// TwinCAT 3 PLC project CamerasTCP_Drivers
// ProgramVersion: 3.1.4026.19
// libraries:
//   Tc2_SerialCom, * (Beckhoff Automation GmbH)
//   Tc2_Standard, * (Beckhoff Automation GmbH)
//   Tc2_System, * (Beckhoff Automation GmbH)
//   Tc2_TcpIp, * (Beckhoff Automation GmbH)
//   Tc2_Utilities, * (Beckhoff Automation GmbH)
// project tree:
//   DUTs/ E_STRING_ExtrMode.TcDUT (not stored), E_TCPIP_RequescCommand.TcDUT, E_TCPIP_SEND_STATE.TcDUT, E_TCPIP_State.TcDUT, T_LongSTRING.TcDUT (not stored)
//   DUTs/NewModel/CameraImage/ E_CAMERA_State.TcDUT, ST_CAMERA_CodeData.TcDUT, ST_CAMERA_ImageData.TcDUT, ST_CAMERA_TriggerID.TcDUT, ST_GS1_AI.TcDUT
//   DUTs/NewModel/ E_CAMERA_Name.TcDUT, ST_CAMERA_Evaluation.TcDUT
//   DUTs/NewModel/Main Struct/Config/ E_CAMERA_CodeType.TcDUT, E_CAMERA_DeviceType.TcDUT, E_CAMERA_Vendor.TcDUT, ST_CAMERA_Options.TcDUT
//   DUTs/NewModel/Main Struct/Control/ ST_CAMERA_BrowseCtrl.TcDUT, ST_CAMERA_Mapping.TcDUT
//   DUTs/NewModel/Main Struct/Status/ E_CAMERA_Status.TcDUT, ST_CAMERA_BrowserStatus.TcDUT, ST_CAMERA_IN.TcDUT, ST_CAMERA_OpState.TcDUT, ST_CAMERA_OUT.TcDUT, ST_CAMERA_Performance.TcDUT
//   DUTs/NewModel/Main Struct/ ST_CAMERA_Config.TcDUT, ST_CAMERA_Ctrl.TcDUT, ST_CAMERA_Status.TcDUT
//   DUTs/Test_DUTs/ ST_DuplicateInfo.TcDUT (not stored), ST_LAB_CaseData.TcDUT, ST_LAB_OuterData.TcDUT, ST_LAB_PackData.TcDUT (not stored)
//   DUTs/USED/ E_SCANNER_CodeType.TcDUT (not stored), E_SCANNER_DeviceType.TcDUT (not stored), E_SCANNER_State.TcDUT (not stored), E_SCANNER_Vendor.TcDUT (not stored), ST_SCANNER.TcDUT, ST_SCANNER_ApplicationIdentifier.TcDUT (not stored), ST_SCANNER_CameraMap.TcDUT (not stored), ST_SCANNER_CodeData.TcDUT (not stored), ST_SCANNER_Config.TcDUT (not stored), ST_SCANNER_Evaluation.TcDUT (not stored), ST_SCANNER_ImageData.TcDUT (not stored), ST_SCANNER_ManualCtrl.TcDUT (not stored), ST_SCANNER_OpState.TcDUT (not stored), ST_SCANNER_Options.TcDUT (not stored), ST_SCANNER_Performance.TcDUT (not stored), ST_SCANNER_TriggerID.TcDUT (not stored)
//   GVLs/ gConstants.TcGVL (not stored), GVL.TcGVL, GVL_HIKROBOT_COMMANDS.TcGVL (not stored), GVL_test.TcGVL
//   / PlcTask.TcTTO
//   POUs/Addtionals/ FB_PulseGenerator_Sync.TcPOU (not stored), PRG_ButtonsHandler.TcPOU
//   POUs/CAMERAS/ FB_SCANNER_HikrobotEXT.TcPOU, F_CREATE_MESSAGE.TcPOU (not stored)
//   POUs/ MAIN.TcPOU, PRG_HikrobotHandler.TcPOU
//   POUs/NewModel/ FB_CAMERA_Omron.TcPOU, FB_CAMERA_HIKROBOT.TcPOU
//   POUs/SOFTWARE_lib/TCP FBs/ FB_TCP_ClientPortCtrl.TcPOU, FB_TCP_ClientPortCtrl_V2.TcPOU, FB_TCP_CloseAllPorts.TcPOU, FB_TCP_ReceiveData_V2.TcPOU, FB_TCP_ReceiveLongString.TcPOU (not stored), FB_TCP_ReceiveString.TcPOU (not stored), FB_TCP_SendData.TcPOU, FB_TCP_ServerPortCtrl.TcPOU
//   POUs/StringFBs/ FB_ExtractAnyString.TcPOU
//   POUs/Tests/ FB_FIND_OuterDuplicates.TcPOU, IO_logic.TcPOU (not stored), Outer_IN_Case_Duplicat.TcPOU, PRG_Test.TcPOU
// real-time tasks:
//   TASK PlcTask: cycle T#10ms, priority 20, ADS port 350
// motion (NC):
//   TASK NC-Task 1 SAF: cycle T#2ms, priority 4, ADS port 501
//   TASK NC-Task 1 SVB: cycle T#10ms, priority 8, ADS port 511
//   AXIS Axis 1 (id 1)
//     OtherSettings: AllowMotionCmdToSlave=true
//     encoder EncType=4
//       EncPara: MaxCount=#x0000ffff
//         Inc: RefSoftSyncMask=#x0000ffff
//     drive DrvType=24
//       Analog: TorqueSetpointScale=10, ScaleFactorActTorque=0.1
//       TimeComp: TaskDelayCycles=1
//     controller CtrType=1
//       CtrPara: PriorControlFactor=1
//         Observer: BandWidth=20
//   AXIS Axis 2 (id 2)
//     OtherSettings: AllowMotionCmdToSlave=true
//     encoder EncType=4
//       EncPara: MaxCount=#x0000ffff
//         Inc: RefSoftSyncMask=#x0000ffff
//     drive DrvType=24
//       Analog: TorqueSetpointScale=10, ScaleFactorActTorque=0.1
//       TimeComp: TaskDelayCycles=1
//     controller CtrType=1
//       CtrPara: PriorControlFactor=1
//         Observer: BandWidth=20
//   AXIS Axis 3 (id 3)
//     OtherSettings: AllowMotionCmdToSlave=true
//     encoder EncType=19
//       EncPara: MaxCount=#xffffffff
//     drive DrvType=16
//       DrvPara: MaxCount=#xffffffff
//         Analog: TorqueSetpointScale=10, ScaleFactorActTorque=0.1
//         TimeComp: TaskDelayCycles=1
//     controller CtrType=1
//       CtrPara: PriorControlFactor=1
//         Observer: BandWidth=20
//   AXIS Axis 4 (id 4)
//     OtherSettings: AllowMotionCmdToSlave=true
//     encoder EncType=4
//       EncPara: MaxCount=#x0000ffff
//         Inc: RefSoftSyncMask=#x0000ffff
//     drive DrvType=24
//       Analog: TorqueSetpointScale=10, ScaleFactorActTorque=0.1
//       TimeComp: TaskDelayCycles=1
//     controller CtrType=1
//       CtrPara: PriorControlFactor=1
//         Observer: BandWidth=20
//   AXIS Axis 5 (id 5)
//     OtherSettings: AllowMotionCmdToSlave=true
//     encoder EncType=4
//       EncPara: MaxCount=#x0000ffff
//         Inc: RefSoftSyncMask=#x0000ffff
//     drive DrvType=24
//       Analog: TorqueSetpointScale=10, ScaleFactorActTorque=0.1
//       TimeComp: TaskDelayCycles=1
//     controller CtrType=1
//       CtrPara: PriorControlFactor=1
//         Observer: BandWidth=20
//   AXIS Axis 6 (id 6)
//     OtherSettings: AllowMotionCmdToSlave=true
//     encoder EncType=19
//       EncPara: MaxCount=#xffffffff
//     drive DrvType=16
//       DrvPara: MaxCount=#xffffffff
//         Analog: TorqueSetpointScale=10, ScaleFactorActTorque=0.1
//         TimeComp: TaskDelayCycles=1
//     controller CtrType=1
//       CtrPara: PriorControlFactor=1
//         Observer: BandWidth=20
//   AXIS Axis 7 (id 7)
//     OtherSettings: AllowMotionCmdToSlave=true
//     encoder EncType=4
//       EncPara: MaxCount=#x0000ffff
//         Inc: RefSoftSyncMask=#x0000ffff
//     drive DrvType=24
//       Analog: TorqueSetpointScale=10, ScaleFactorActTorque=0.1
//       TimeComp: TaskDelayCycles=1
//     controller CtrType=1
//       CtrPara: PriorControlFactor=1
//         Observer: BandWidth=20
//   AXIS Axis 8 (id 8)
//     OtherSettings: AllowMotionCmdToSlave=true
//     encoder EncType=4
//       EncPara: MaxCount=#x0000ffff
//         Inc: RefSoftSyncMask=#x0000ffff
//     drive DrvType=24
//       Analog: TorqueSetpointScale=10, ScaleFactorActTorque=0.1
//       TimeComp: TaskDelayCycles=1
//     controller CtrType=1
//       CtrPara: PriorControlFactor=1
//         Observer: BandWidth=20
//   AXIS Axis 9 (id 9)
//     OtherSettings: AllowMotionCmdToSlave=true
//     encoder EncType=19
//       EncPara: MaxCount=#xffffffff
//     drive DrvType=16
//       DrvPara: MaxCount=#xffffffff, DriveControlDWord=#x00020000
//         Analog: TorqueSetpointScale=10, ScaleFactorActTorque=0.1
//         TimeComp: TaskDelayCycles=1
//     controller CtrType=1
//       CtrPara: PriorControlFactor=1
//         Observer: BandWidth=20
//   AXIS Axis 10 (id 10)
//     OtherSettings: AllowMotionCmdToSlave=true
//     encoder EncType=4
//       EncPara: MaxCount=#x0000ffff
//         Inc: RefSoftSyncMask=#x0000ffff
//     drive DrvType=24
//       Analog: TorqueSetpointScale=10, ScaleFactorActTorque=0.1
//       TimeComp: TaskDelayCycles=1
//     controller CtrType=1
//       CtrPara: PriorControlFactor=1
//         Observer: BandWidth=20
//   AXIS Axis 11 (id 11)
//     OtherSettings: AllowMotionCmdToSlave=true
//     encoder EncType=4
//       EncPara: MaxCount=#x0000ffff
//         Inc: RefSoftSyncMask=#x0000ffff
//     drive DrvType=24
//       Analog: TorqueSetpointScale=10, ScaleFactorActTorque=0.1
//       TimeComp: TaskDelayCycles=1
//     controller CtrType=1
//       CtrPara: PriorControlFactor=1
//         Observer: BandWidth=20
//   AXIS Axis 12 (id 12)
//     OtherSettings: AllowMotionCmdToSlave=true
//     encoder EncType=19
//       EncPara: MaxCount=#xffffffff
//     drive DrvType=16
//       DrvPara: MaxCount=#xffffffff
//         Analog: TorqueSetpointScale=10, ScaleFactorActTorque=0.1
//         TimeComp: TaskDelayCycles=1
//     controller CtrType=1
//       CtrPara: PriorControlFactor=1
//         Observer: BandWidth=20
// I/O:
//   DEVICE Device 1 (EtherCAT) (disabled), AmsNetId 192.168.1.11.2.1
//     Term 1 (EK1100)
//     Term 9 (EK1100) [EK1100 EtherCAT Coupler (2A E-Bus)]
//       Term 10 (EL7031-0030)
//       Term 11 (EL6070-0033)
//       Term 12 (EL7031-0030)
//       Term 17 (EL9011)
//     Term 13 (EK1818)
// variable links:
//   (this object) <-> Device 1 (EtherCAT)/Term 9 (EK1100)/Term 10 (EL7031-0030)
//     Drive/Inputs/In/nState1 @bit 3 <-> STM Status/Status/Error
//     Drive/Inputs/In/nState1 @bit 5 <-> STM Status/Status/Moving negative
//     Drive/Inputs/In/nState1 @bit 4 <-> STM Status/Status/Moving positive
//     Drive/Inputs/In/nState1 @bit 1 <-> STM Status/Status/Ready
//     Drive/Inputs/In/nState1 <-> STM Status/Status/Ready to enable
//     Drive/Inputs/In/nState1 @bit 6 <-> STM Status/Status/Torque reduced
//     Drive/Inputs/In/nState1 @bit 2 <-> STM Status/Status/Warning
//     Drive/Inputs/In/nState2 @bit 3 <-> STM Status/Status/Digital input 1
//     Drive/Inputs/In/nState2 @bit 4 <-> STM Status/Status/Digital input 2
//     Drive/Inputs/In/nState2 @bit 5 <-> STM Status/Status/Sync error
//     Drive/Inputs/In/nState2 @bit 7 <-> STM Status/Status/TxPDO Toggle
//     Drive/Inputs/In/nState4 @bit 1 <-> WcState/InputToggle
//     Drive/Inputs/In/nState4 <-> WcState/WcState
//     Drive/Outputs/Out/nCtrl1 <-> STM Control/Control/Enable
//     Drive/Outputs/Out/nCtrl1 @bit 2 <-> STM Control/Control/Reduce torque
//     Drive/Outputs/Out/nCtrl1 @bit 1 <-> STM Control/Control/Reset
//     Drive/Outputs/Out/nDataOut2[0] <-> STM Velocity/Velocity
//     Enc/Inputs/In/nDataIn1[0] <-> ENC Status compact/Counter value
//     Enc/Inputs/In/nDataIn2[0] <-> ENC Status compact/Latch value
//     Enc/Inputs/In/nState1 @bit 4 <-> ENC Status compact/Status/Counter overflow
//     Enc/Inputs/In/nState1 @bit 3 <-> ENC Status compact/Status/Counter underflow
//     Enc/Inputs/In/nState1 @bit 1 <-> ENC Status compact/Status/Latch extern valid
//     Enc/Inputs/In/nState1 @bit 2 <-> ENC Status compact/Status/Set counter done
//     Enc/Inputs/In/nState2 @bit 4 <-> ENC Status compact/Status/Status of extern latch
//     Enc/Inputs/In/nState2 @bit 5 <-> ENC Status compact/Status/Sync error
//     Enc/Inputs/In/nState2 @bit 7 <-> ENC Status compact/Status/TxPDO Toggle
//     Enc/Inputs/In/nState4 @bit 1 <-> WcState/InputToggle
//     Enc/Inputs/In/nState4 <-> WcState/WcState
//     Enc/Outputs/Out/nCtrl1 @bit 3 <-> ENC Control compact/Control/Enable latch extern on negative edge
//     Enc/Outputs/Out/nCtrl1 @bit 1 <-> ENC Control compact/Control/Enable latch extern on positive edge
//     Enc/Outputs/Out/nCtrl1 @bit 2 <-> ENC Control compact/Control/Set counter
//     Enc/Outputs/Out/nDataOut1[0] <-> ENC Control compact/Set counter value
//   (this object) <-> Device 1 (EtherCAT)/Term 9 (EK1100)/Term 12 (EL7031-0030)
//     Drive/Inputs/In/nState1 @bit 3 <-> STM Status/Status/Error
//     Drive/Inputs/In/nState1 @bit 5 <-> STM Status/Status/Moving negative
//     Drive/Inputs/In/nState1 @bit 4 <-> STM Status/Status/Moving positive
//     Drive/Inputs/In/nState1 @bit 1 <-> STM Status/Status/Ready
//     Drive/Inputs/In/nState1 <-> STM Status/Status/Ready to enable
//     Drive/Inputs/In/nState1 @bit 6 <-> STM Status/Status/Torque reduced
//     Drive/Inputs/In/nState1 @bit 2 <-> STM Status/Status/Warning
//     Drive/Inputs/In/nState2 @bit 3 <-> STM Status/Status/Digital input 1
//     Drive/Inputs/In/nState2 @bit 4 <-> STM Status/Status/Digital input 2
//     Drive/Inputs/In/nState2 @bit 5 <-> STM Status/Status/Sync error
//     Drive/Inputs/In/nState2 @bit 7 <-> STM Status/Status/TxPDO Toggle
//     Drive/Inputs/In/nState4 @bit 1 <-> WcState/InputToggle
//     Drive/Inputs/In/nState4 <-> WcState/WcState
//     Drive/Outputs/Out/nCtrl1 <-> STM Control/Control/Enable
//     Drive/Outputs/Out/nCtrl1 @bit 2 <-> STM Control/Control/Reduce torque
//     Drive/Outputs/Out/nCtrl1 @bit 1 <-> STM Control/Control/Reset
//     Drive/Outputs/Out/nDataOut2[0] <-> STM Velocity/Velocity
//     Enc/Inputs/In/nDataIn1[0] <-> ENC Status compact/Counter value
//     Enc/Inputs/In/nDataIn2[0] <-> ENC Status compact/Latch value
//     Enc/Inputs/In/nState1 @bit 4 <-> ENC Status compact/Status/Counter overflow
//     Enc/Inputs/In/nState1 @bit 3 <-> ENC Status compact/Status/Counter underflow
//     Enc/Inputs/In/nState1 @bit 1 <-> ENC Status compact/Status/Latch extern valid
//     Enc/Inputs/In/nState1 @bit 2 <-> ENC Status compact/Status/Set counter done
//     Enc/Inputs/In/nState2 @bit 4 <-> ENC Status compact/Status/Status of extern latch
//     Enc/Inputs/In/nState2 @bit 5 <-> ENC Status compact/Status/Sync error
//     Enc/Inputs/In/nState2 @bit 7 <-> ENC Status compact/Status/TxPDO Toggle
//     Enc/Inputs/In/nState4 @bit 1 <-> WcState/InputToggle
//     Enc/Inputs/In/nState4 <-> WcState/WcState
//     Enc/Outputs/Out/nCtrl1 @bit 3 <-> ENC Control compact/Control/Enable latch extern on negative edge
//     Enc/Outputs/Out/nCtrl1 @bit 1 <-> ENC Control compact/Control/Enable latch extern on positive edge
//     Enc/Outputs/Out/nCtrl1 @bit 2 <-> ENC Control compact/Control/Set counter
//     Enc/Outputs/Out/nDataOut1[0] <-> ENC Control compact/Set counter value
//   (this object) <-> Device 1 (EtherCAT)/Term 13 (EK1818)/Term 14 (EL7211-9014)
//     Drive/Inputs/In/nDcOutputTime <-> InfoData/DcOutputShift
//     Drive/Inputs/In/nState1 <-> DRV Statusword/Statusword
//     Drive/Inputs/In/nState2 <-> DRV Statusword/Statusword @bit 8
//     Drive/Inputs/In/nState4 @bit 1 <-> WcState/InputToggle
//     Drive/Inputs/In/nState4 <-> WcState/WcState
//     Drive/Outputs/Out/nCtrl1 <-> DRV Controlword/Controlword
//     Drive/Outputs/Out/nCtrl2 <-> DRV Controlword/Controlword @bit 8
//     Drive/Outputs/Out/nDataOut2 <-> DRV Target velocity/Target velocity
//     Enc/Inputs/In/nDataIn1 <-> FB Position/Position
//     Enc/Inputs/In/nDcInputTime <-> InfoData/DcInputShift
//     Enc/Inputs/In/nState4 @bit 1 <-> WcState/InputToggle
//     Enc/Inputs/In/nState4 <-> WcState/WcState

CONFIGURATION CamerasTCP_Drivers
    RESOURCE PLC ON TwinCAT3
        TASK PlcTask(INTERVAL := T#10ms, PRIORITY := 20);
        PROGRAM MAIN WITH PlcTask : MAIN;
    END_RESOURCE
END_CONFIGURATION

// ---- DUTs/E_TCPIP_RequescCommand.TcDUT
{attribute 'qualified_only'}
{attribute 'strict'}
{attribute 'to_string'}
TYPE E_TCPIP_RequescCommand :
(
	NONE,					(* No request to send *)
	SetRunMode,				(* Set run mode, 0 - Normal, 1 - Raw, 2 - Test *)
	SetAcq,					(* Set acquisition mode, 0 - Stop acq, 1 - Start acq *)
	GetUserCur,
	HeartbeatCheck			
);
END_TYPE

// ---- DUTs/E_TCPIP_SEND_STATE.TcDUT
{attribute 'qualified_only'}
{attribute 'strict'}
{attribute 'to_string'}
TYPE E_TCPIP_SEND_STATE :
(
	IDLE,
	CONNECT,
	SEND,
	RECEIVE,
	DISCONNECT,
	DONE,
	CONN_RESET,
	HEARTBEAT_CHECK,
	ERROR
);
END_TYPE

// ---- DUTs/E_TCPIP_State.TcDUT
{attribute 'qualified_only'}
{attribute 'strict'}
{attribute 'to_string'}
TYPE E_TCPIP_State :
(
	E_TCPIP_IDLE,
	E_TCPIP_CONNECT,
	E_TCPIP_SEND,
	E_TCPIP_RECEIVE,
	E_TCPIP_DISCONNECT,
	E_TCPIP_CLOSEALL,
	E_TCPIP_DONE
);
END_TYPE

// ---- DUTs/NewModel/CameraImage/E_CAMERA_State.TcDUT
{attribute 'qualified_only'}
{attribute 'strict'}
TYPE E_CAMERA_State :
(
	IDLE,
	CONNECT,
	SEND,
	RECEIVE,
	DISCONNECT,
	//CHECKOS,
	BROWSEDIAG,
	BROWSELIVE,
	IMAGE,
	DECODE,
	HEARTBEAT,
	DONE
);
END_TYPE

// ---- DUTs/NewModel/CameraImage/ST_CAMERA_CodeData.TcDUT
TYPE ST_CAMERA_CodeData :
STRUCT
	nScannerIndex		: INT;			(* scanner index when an array of scanners is used *)
	sDataString			: T_MaxString;	(* data string read from code *)
	eCodeType			: E_CAMERA_CodeType;	(* code type *)
	fOverallGrade		: LREAL;		(* overall grade of code *)
	fXPos				: LREAL;		(* X position of centre of code *)
	fYPos				: LREAL;		(* Y position of centre of code *)
	fAngle				: LREAL;		(* angle of code *)
	fCellSize			: LREAL;		(* cell size *)
	fSymbolContrast		: LREAL;		(* symbol contrast *)
	nEvaluation			: INT;			(* general code quality evaluatio*)
	fUnusedErrCorr		: LREAL;		(* unused error correction *)
	nProgramNo			: BYTE;			(* program number *)
END_STRUCT
END_TYPE

// ---- DUTs/NewModel/CameraImage/ST_CAMERA_ImageData.TcDUT
TYPE ST_CAMERA_ImageData :
STRUCT
	nCodesRead		: INT;
	tScanTime		: TIME;		(* image cycle time (including image acquisition time and decode time) *)
	sDecodeStatus	: T_MaxString;
	stTriggerID		: ST_CAMERA_TriggerID;
	aCodeData		: ARRAY[1..cMAX_CAMERA_PROG_NUMBER] OF ST_CAMERA_CodeData;
END_STRUCT
END_TYPE

// ---- DUTs/NewModel/CameraImage/ST_CAMERA_TriggerID.TcDUT
TYPE ST_CAMERA_TriggerID :
STRUCT
	nTriggerID			: UDINT;
	nScanNo				: INT := 1;
	nScannerIndex		: INT := 1;
END_STRUCT
END_TYPE

// ---- DUTs/NewModel/CameraImage/ST_GS1_AI.TcDUT
TYPE ST_GS1_AI :
STRUCT
	sAI			: STRING(4);
	bFixed		: BOOL;
	nLength		: UINT;
END_STRUCT
END_TYPE

// ---- DUTs/NewModel/E_CAMERA_Name.TcDUT
{attribute 'qualified_only'}
//{attribute 'strict'}
TYPE E_CAMERA_Name :
(
	CAM01		:= 1,
	CAM02		:= 2,
	CAM03		:= 3,
	CAM04		:= 4,
	CAM05		:= 5,
	CAM06		:= 6,
	CAM07		:= 7,
	CAM08		:= 8,
	CAM09		:= 9,
	CAM10		:= 10,
	CAM11		:= 11,
	CAM12		:= 12
);
END_TYPE

// ---- DUTs/NewModel/Main Struct/Config/E_CAMERA_CodeType.TcDUT
{attribute 'qualified_only'}
//{attribute 'strict'}
TYPE E_CAMERA_CodeType :
(
	NONE 		:= 0,
	OCR			:= 7,
	DATAMARTIX	:= 10,
	QR			:= 11,
	DOTCODE		:= 14,
	CODE128		:= 20,
	ITF14		:= 24,
	EAN13		:= 27,
	EAN8		:= 28,
	UNKNOWN		:= 99
);
END_TYPE

// ---- DUTs/NewModel/Main Struct/Config/E_CAMERA_DeviceType.TcDUT
{attribute 'qualified_only'}
//{attribute 'strict'}
TYPE E_CAMERA_DeviceType :    (*tAcquisitionTime - to be secured*)
(
	NONE,
	MV420_F,			//F -> Full resolution
	MV420_H,			//H -> Half resolution
	MV440SR_F,
	MV440SR_H,
	MV440HR_F,
	MV440HR_H,
	MV440UR_F,
	MV440UR_H,
	MV540S_F,
	MV540S_H,
	MV540H_F,
	MV540H_H,
	MV560U_F,
	MV560U_H,
	V430F	(*Omron*)

);
END_TYPE

// ---- DUTs/NewModel/Main Struct/Config/E_CAMERA_Vendor.TcDUT
{attribute 'qualified_only'}
{attribute 'strict'}
TYPE E_CAMERA_Vendor :
(
	SIEMENS		:= 1,
	OMRON 		:= 2,
	KEYENCE		:= 3,
	COGNEX		:= 4,
	HIKROBOT	:= 5
);
END_TYPE

// ---- DUTs/NewModel/Main Struct/Config/ST_CAMERA_Options.TcDUT
TYPE ST_CAMERA_Options :
STRUCT
	eScannerType			: E_CAMERA_DeviceType;
	eExpectedType			: E_CAMERA_CodeType;
	bUseExternalLight		: BOOL;
	nLightingIntensity		: INT;
	nDisplayDelayConfig		: BOOL;

	nImageBuffer			: INT := 1;
	nExpectedResp			: INT := 1;
	
	aCameraWarningLevel		: INT := 90;
	sFC1ReplacmentChar		: T_Char;
END_STRUCT
END_TYPE

// ---- DUTs/NewModel/Main Struct/Control/ST_CAMERA_BrowseCtrl.TcDUT
TYPE ST_CAMERA_BrowseCtrl :
STRUCT
	bBrowseLive			: BOOL;	
	bBrowseDiag			: BOOL;
END_STRUCT
END_TYPE

// ---- DUTs/NewModel/Main Struct/Control/ST_CAMERA_Mapping.TcDUT
TYPE ST_CAMERA_Mapping :
STRUCT
	nIndex				: INT;
	nReqProgram			: BYTE;
	aPackPos			: ARRAY[1..5, 1..cMAX_CAMERA_PROG_NUMBER] OF BYTE;
	aTargetBuffer		: ARRAY[1..5] OF BYTE;

END_STRUCT
END_TYPE

// ---- DUTs/NewModel/Main Struct/Status/E_CAMERA_Status.TcDUT
{attribute 'qualified_only'}
{attribute 'strict'}

TYPE E_CAMERA_Status :
(
			
	DIABLED 		:= 0,		//0 = Grey, disabled OR offline
	CONFIG			:= 1,		//1 = Blue, configuration mode active
	ALARM			:= 2,		//2 = Red, alarm active or comms loss
	EXTERNALOFF		:= 3,		//3 = Orange, external condition off
	WARNING			:= 4,		//4 = Yellow, warning active
	OERATIONAL		:= 5		//5 = Green, operational	
);
END_TYPE

// ---- DUTs/NewModel/Main Struct/Status/ST_CAMERA_BrowserStatus.TcDUT
TYPE ST_CAMERA_BrowserStatus :
STRUCT
	bBrowseLiveActive			: BOOL;	
	bBrowseDiagActive			: BOOL;
END_STRUCT
END_TYPE

// ---- DUTs/NewModel/Main Struct/Status/ST_CAMERA_IN.TcDUT
TYPE ST_CAMERA_IN :
STRUCT
	stTriggerID			: ST_CAMERA_TriggerID;	
	stBrowserStatus		: ST_CAMERA_BrowserStatus;
	
END_STRUCT
END_TYPE

// ---- DUTs/NewModel/Main Struct/Status/ST_CAMERA_OpState.TcDUT
TYPE ST_CAMERA_OpState :
STRUCT
	nStatusByte			: BYTE;
	nErrorCode			: UDINT;
	nWarningCode		: UDINT;

	bAcceptTrigger		: BOOL;
	bCodeChangeActive	: BOOL;
	nActiveTriggers		: INT;

	bTCPComsLockedUp	: BOOL;

END_STRUCT
END_TYPE

// ---- DUTs/NewModel/Main Struct/Status/ST_CAMERA_OUT.TcDUT
TYPE ST_CAMERA_OUT :
STRUCT
	bDone								: BOOL;			(* TRUE = code scan complete *)
	bBusy								: BOOL;			(* TRUE = code scan in progress *)
	bError								: BOOL;			(* TRUE = code scan error *)

	bReady								: BOOL;			(* TRUE = scanner port connected *)
	bEnableActive						: BOOL;
	nTriggerCounter						: UDINT;

	nActiveProgram						: BYTE;			(* active program *)
	stOpState							: ST_CAMERA_OpState;	(* operating state values *)
	
	sCodeStatus							: T_MaxString;				(* image status string *)
	sCurrentCodeRead					: T_MaxString;
	aLast10CodesRead					: ARRAY[1..10]  OF T_MaxString;
	stImageData							: ST_CAMERA_ImageData;		(* image data structure *)
	stReadPerformance					: ST_CAMERA_Performance;
	
	eSocketState						: E_SocketConnectionState;	(* TCP socket connection state *)
	
	bLastBarcodeValid					: BOOL;
	sLastStatus							: T_MaxString;
	
	bCameraTrigger						: BOOL;			(* TRG signal to camera - physical output *)
	bLightTrigger						: BOOL;			(* TRG signal to ext light - physical output *)

END_STRUCT
END_TYPE

// ---- DUTs/NewModel/Main Struct/Status/ST_CAMERA_Performance.TcDUT
TYPE ST_CAMERA_Performance :
STRUCT
	tLastDiff 		: TIME;
	tAverageDiff 	: TIME;
	arrTimeDiff 	: ARRAY[0..9] OF TIME;
END_STRUCT
END_TYPE

// ---- DUTs/NewModel/Main Struct/ST_CAMERA_Config.TcDUT
TYPE ST_CAMERA_Config :     //ST_SCANNER_Config
STRUCT
	sDeviceName				: STRING(30) := 'Camera';
	bDisableCameraUse		: BOOL;

	stCameraIP				: ST_TCPIP_AddressPort;
	stOptions				: ST_CAMERA_Options;
	bDontParseAsGS1			: BOOL;
	
	tTimeOut				: TIME := T#3S;
	eCameraVendor			: E_CAMERA_Vendor;
	
END_STRUCT
END_TYPE

// ---- DUTs/NewModel/Main Struct/ST_CAMERA_Ctrl.TcDUT
TYPE ST_CAMERA_Ctrl :    //ST_SCANNER_CameraMap
STRUCT
	bProcessNewCode		: BOOL;
	bManualTrigger		: BOOL;
	bConfigMode			: BOOL;	
	bResetStats			: BOOL;	
	
	stBrowseCtrl		: ST_CAMERA_BrowseCtrl;
	stCameraMap			: ST_CAMERA_Mapping;
END_STRUCT
END_TYPE

// ---- DUTs/NewModel/Main Struct/ST_CAMERA_Status.TcDUT
TYPE ST_CAMERA_Status :   //ST_SCANNER
STRUCT
	
	nStatus	: BYTE;
	eStatus	: E_CAMERA_Status;
	
	I		: ST_CAMERA_IN;
	Q		: ST_CAMERA_OUT;
	
END_STRUCT
END_TYPE

// ---- DUTs/NewModel/ST_CAMERA_Evaluation.TcDUT
TYPE ST_CAMERA_Evaluation :
STRUCT
	nTotalReads			: UDINT;
	nReadCodes			: UDINT;
	nNOKCodes			: UDINT;

	nGoodCodes			: UDINT;
	nFairCodes			: UDINT;
	nPoorCodes			: UDINT;

	fReadEfficiency			: LREAL;
	fNOKEfficiency			: LREAL;

	fGoodEfficiency		: LREAL;
	fFairEfficiency			: LREAL;
	fPoorEfficiency			: LREAL;

END_STRUCT
END_TYPE

// ---- DUTs/Test_DUTs/ST_LAB_CaseData.TcDUT
TYPE ST_LAB_CaseData :
STRUCT
	aOuters		: ARRAY[1..3] OF ST_LAB_OuterData;
END_STRUCT
END_TYPE

// ---- DUTs/Test_DUTs/ST_LAB_OuterData.TcDUT
TYPE ST_LAB_OuterData :
STRUCT
	sOuterCode			: T_MaxString;
	nOutersStatus		: INT;
	nOuterRejectID		: UINT;
	
	aPacks				: ARRAY[1..3] OF ST_LAB_PackData;
END_STRUCT
END_TYPE

// ---- DUTs/USED/ST_SCANNER.TcDUT
TYPE ST_SCANNER :
STRUCT
	bReady								: BOOL;
	nState								: BYTE;
	bLastBarcodeValid					: BOOL;
(**)	strLastCodeRead					: T_MaxString;
(**)	strLastBarcode						: STRING(253);	(*zenon*)
	strCurrentCodeRead					: T_MaxString;
	aLast10CodesRead					: ARRAY[1..10]  OF T_MaxString;
	strLastStatus						: T_MaxString;
	nTriggerCounter						: UDINT;
	sManualCtrlScanner					: ST_SCANNER_ManualCtrl;
(**)(*	sSStats							: ST_SCANNER_Statistics;*)
	sScannerOpState						: ST_SCANNER_OpState;
	sImageData							: ST_SCANNER_ImageData;
	bEnableActive						: BOOL;
	nActiveProgram						: BYTE;
	bAcceptTrigger						: BOOL;
	stTriggerID							: ST_SCANNER_TriggerID;
	eSocketState						: E_SocketConnectionState;
	sReadPerformance					: ST_SCANNER_Performance;
END_STRUCT
END_TYPE

// ---- GVLs/GVL.TcGVL
{attribute 'qualified_only'}
VAR_GLOBAL
	bTriggerButton		AT %I* : BOOL;			
	bTriggerOutput		AT %Q* : BOOL;		


	// Hikrobot Control Commands

	aHikrobotCtrlCommands				: ARRAY[1..20] OF STRING(40) :=[
		(*start user params 0*) 		'<Set,UserStart,0>',
		(*start user params 1*) 		'<Set,UserStart,1>',
		(*start user params 2*) 		'<Set,UserStart,2>',
		(*execute self adjustement*) 	'<Exec,Tune>',
		(*start reading codes*) 		'<Set,Acq,1><Set,UserStart,3>',
		(*stop reading codes*) 			'<Set,Acq,0>',
		(*camera reboot*) 				'<Exec,Reboot>',
		(*camera reboot*) 				'<Get,RunMode>',
		(*camera reboot*) 				'<Set,RunMode,2>',
		(*camera reboot*) 				'<Set,RunMode,0>'
];


	aTCPxStrings						: ARRAY[0..20] OF T_MaxString;

END_VAR

// ---- GVLs/GVL_test.TcGVL
{attribute 'qualified_only'}
VAR_GLOBAL
	
	//aCase	: ARRAY[1..3] OF ST_LAB_OuterData ;
	stCase		:	ST_LAB_CaseData; 
	stCaseFull	:	ST_LAB_CaseData; 

	
// 	aInputArray		: ARRAY[1..3, 1..3] OF T_MaxString := [ 
// 	['PACK01OUTER1', 'PACK02OUTER1', 'PACK03OUTER1'],
// 	['PACK01OUTER2', 'PACK02OUTER2', 'PACK03OUTER2'],
// 	['PACK01OUTER3', 'PACK02OUTER3', 'PACK03OUTER3']
// 	];

END_VAR

// ---- POUs/MAIN.TcPOU
PROGRAM MAIN
VAR
	
	
END_VAR


//fbSiemensCameraMV5xCtrl();

//PRG_Test();
PRG_ButtonsHandler();

//IO_logic();

PRG_HikrobotHandler();

	
//Outer_IN_Case_Duplicat();

END_PROGRAM

// ---- POUs/Addtionals/PRG_ButtonsHandler.TcPOU
PROGRAM PRG_ButtonsHandler
VAR
	rTrig			: R_TRIG;
	tTimer			: TOF;
	tTriggerTime	: TIME := T#100MS;
	bTimerOn		: BOOL;
	iIteration		: INT;
	
	fbTON			: TON;
	fbTOF			: TOF;
	bOut			: BOOL;
	bEnable			: BOOL;
END_VAR


rTrig(CLK:= GVL.bTriggerButton);

tTimer(IN:= bTimerOn, PT:= tTriggerTime);

IF rTrig.Q THEN
	bTimerOn := TRUE;	
ELSIF tTimer.ET = T#0S THEN
	bTimerOn := FALSE;
END_IF

//petla strzelania 10 fotek


fbTON(IN := NOT bOut, PT := T#200MS);
fbTOF(IN := bOut, PT := T#100MS); 

IF rTrig.Q THEN
	bEnable := TRUE;
END_IF

IF bEnable THEN
	IF fbTON.Q THEN                // Po 500 ms OFF -> załącz
		bOut := TRUE;
		iIteration := iIteration + 1;
	ELSIF fbTOF.Q THEN             // Po 100 ms ON -> wyłącz
		bOut := FALSE;
	END_IF
	
	IF iIteration > 5 THEN
		iIteration 	:= 0;
		bEnable		:= FALSE;
	END_IF
	
ELSE
	bOut := FALSE;   
	// Reset przy wyłączonym
END_IF

GVL.bTriggerOutput := bOut;	



//GVL.bTriggerOutput := tTimer.Q;

END_PROGRAM

// ---- POUs/PRG_HikrobotHandler.TcPOU
PROGRAM PRG_HikrobotHandler
VAR	
	
	fbHikrobotScannerCtrl			: FB_SCANNER_HikrobotEXT;
	
	// HIKROBOT Inputs
	bEnableReceive					: BOOL;
	bEnableSend						: BOOL;
	strScannerIPAddr				: T_IPv4Addr	:= '192.168.1.45';
	nReceiveScannerPortNo			: UINT			:= 2010;
	nSendScannerPortNo				: UINT			:= 4001;	
	stRequestCommand				: E_TCPIP_RequescCommand; (* tutaj powinna byc strukruta z eRequestCommand plus parametry: 0,1 etc *)
	bSendCommand					: BOOL;
	bExecutedCommandSend			: BOOL;
	
	// HIKROBOT Outputs
	eSocketReceiveState			: E_SocketConnectionState;
	eSocketSendState			: E_SocketConnectionState;
	strTCPRxStringOut			: T_MaxString;
	
	fbExtractAnyString			: FB_ExtractAnyString();
	// Extracted String IN_OUT
	strTCP_HikrobotReceived		: T_MaxString;

END_VAR


fbHikrobotScannerCtrl(
	bEnableReceive:= bEnableReceive, 
	bEnableSend:= bEnableSend, 
	strScannerIPAddr:= strScannerIPAddr, 
	nReceiveScannerPortNo:= nReceiveScannerPortNo, 
	nSendScannerPortNo:= nSendScannerPortNo, 
	stRequestCommand:= stRequestCommand, 
	bSendCommand:= bSendCommand, 
	bExecutedCommandSend:= bExecutedCommandSend, 
	eSocketReceiveState=> eSocketReceiveState, 
	eSocketSendState=> eSocketSendState, 
	strTCPRxStringOut=> strTCP_HikrobotReceived
);

fbExtractAnyString(
	bExtractData:= , 
	nExtractChars:= , 
	sPrefix:= , 
	sSuffix:= , 
	bIgnoreCase:= , 
	eExtractMode:= , 
	sDataString:= strTCP_HikrobotReceived, 
	bStringFound=> , 
	sExtractedString=> , 
	nExtractedStringPos=> , 
	nExtractedStringLen=> , 
	nDataStringLen=> 
);

END_PROGRAM

// ---- POUs/CAMERAS/FB_SCANNER_HikrobotEXT.TcPOU
FUNCTION_BLOCK FB_SCANNER_HikrobotEXT
VAR_INPUT
	bEnableReceive					: BOOL;
	bEnableSend						: BOOL;
	strScannerIPAddr				: T_IPv4Addr;
	nReceiveScannerPortNo			: UINT;
	nSendScannerPortNo				: UINT;	
	stRequestCommand				: E_TCPIP_RequescCommand; (* tutaj powinna byc strukruta z eRequestCommand plus parametry: 0,1 etc *)
	bSendCommand					: BOOL;
	bExecutedCommandSend			: BOOL;
END_VAR

VAR_OUTPUT
	eSocketReceiveState		: E_SocketConnectionState;
	eSocketSendState		: E_SocketConnectionState;
	strTCPRxStringOut		: T_MaxString;
	
END_VAR

VAR
	fbTCPPortCtrl_Receive	: FB_TCP_ClientPortCtrl;
	bReceiveConnected		: BOOL;
	
	fbTCPortCtrl_Send		: FB_TCP_ClientPortCtrl;
	bSendConnected			: BOOL;
	
	fbTCPReceive			: FB_ReceiveString;
	bReceiveExpected		: BOOL;
	fbTCPReceiveAfterSend	: FB_ReceiveString;	
	strTCPRxStringReply		: T_MaxString;
	strTCPRxString			: T_MaxString;
	strTCPRxString_Reply	: T_MaxString;
	ftrigEnable				: F_TRIG;
	bReInitialiseTCP		: BOOL;
	fbTON_TcpTimeout		: TON;
	
	nIndex					: UINT;
	nIndexReply				: UINT;
	nIndex2					: UINT;
	
	/////// send command
	
	fbTCPSend				: FB_SocketSend;
	rTrigSend				: R_TRIG;
	rTrigDataReceived		: R_TRIG;
	rTrigSendCommand		: R_TRIG;
	nCommandNo				: UINT := 1;
	fTrigTCPSendDone		: F_TRIG;
	nSendErrId				: UDINT;
	strTCPCommand			: STRING(20);
	strReplyString			: STRING(20);
	strTCPLastCommand		: STRING(20);
	strLastReplyString		: STRING(20);
	bReplyOK				: BOOL;
	tHeartbeatInterval		: TIME := T#5S;
	eRequestCommand			: E_TCPIP_RequescCommand;
	
	(* SEND SEQUENCE VARIABLE *)
	
	eSendSequenceSTATE		: E_TCPIP_SEND_STATE;
	bSendRequest			: BOOL;
	rTrigSendRequest		: R_TRIG;
END_VAR


Connect();

Receive();

//Send();

Send_Sequence();

ACTION Connect:

(* TCP Receive Socket establish connect *)
fbTCPPortCtrl_Receive(
	bEnable				:= bEnableReceive, 
	strRemoteIPAddr		:= strScannerIPAddr, 
	nRemotePortNo		:= nReceiveScannerPortNo, 
	tReconnectTime		:= T#20S, 
	eSocketState		=> eSocketReceiveState, 
	bError				=> , 
	nErrorID			=>,
	bConnected			=> bReceiveConnected
 );
	
(* TCP Send Socket establish connect *)
fbTCPortCtrl_Send(
	bEnable				:= bEnableSend, 
	strRemoteIPAddr		:= strScannerIPAddr, 
	nRemotePortNo		:= nSendScannerPortNo, 
	tReconnectTime		:= T#20S, 
	eSocketState		=> eSocketSendState, 
	bError				=> , 
	nErrorID			=>, 
	bConnected			=> bSendConnected
);
END_ACTION

ACTION Patch:


IF fbTCPReceive.bDataReceived THEN
	GVL.aTCPxStrings[nIndex] := strTCPRxString;
	nIndex := nIndex + 1;
	strTCPRxString := '';
END_IF
// zeroj tablice otrzymanych stringow	
IF nIndex = 20 THEN
	nIndex := 0;
	FOR nIndex2 := 0 TO 20 DO
		GVL.aTCPxStrings[nIndex2] := '';		
	END_FOR
END_IF
// zeroj tablice odpowiedzi na porcie send
IF nIndexReply = 20 THEN
	nIndexReply := 0;
	FOR nIndex2 := 0 TO 20 DO
		GVL.aTCPxStringsReply[nIndex2] := '';		
	END_FOR
END_IF
END_ACTION

ACTION Receive:

ftrigEnable(CLK := bEnableReceive);
IF ftrigEnable.Q THEN
	strTCPRxString := ''; (* clears input buffer *)
END_IF

(* poll TCP port receive string *)
fbTCPReceive(
	bEnable			:= fbTCPPortCtrl_Receive.bConnected,
	hSocket			:= fbTCPPortCtrl_Receive.hSocket,
	tUpdateTime		:= T#100MS,
	strTCPRxString	:= strTCPRxString
);

//Patch();

IF fbTCPReceive.bDataReceived THEN
	
	strTCPRxStringOut := strTCPRxString;	
	
END_IF
END_ACTION

ACTION Send:

rTrigSend(CLK := bSendCommand);
IF rTrigSend.Q THEN
	strTCPCommand 	:= GVL.aHikrobotCtrlCommands[nCommandNo];	
END_IF

fbTCPSend(
	sSrvNetId	:= '',
	hSocket		:= fbTCPortCtrl_Send.hSocket,
	cbLen		:= TO_UDINT(LEN(strTCPCommand)),
	pSrc		:= ADR(strTCPCommand),
	bExecute	:= rTrigSend.Q,
	tTimeout	:= T#1s
);

(* send data complete *)
fTrigTCPSendDone(CLK := fbTCPSend.bBusy);
(* TCP send complete *)

IF fbTCPSend.bError = TRUE THEN
	nSendErrId := fbTCPSend.nErrId;
ELSE
	nSendErrId := 0;	
END_IF

IF fTrigTCPSendDone.Q = TRUE THEN

	(* clear strTCPCommand *)
	strTCPCommand := '';

	(* close off fbSendTCPData *)
	fbTCPSend(bExecute := FALSE);
END_IF


// expece response after sending command
fbTCPReceiveAfterSend(
	bEnable			:= bSendCommand AND fbTCPortCtrl_Send.bConnected,
	hSocket			:= fbTCPortCtrl_Send.hSocket,
	tUpdateTime		:= T#100MS,
	strTCPRxString	:= strTCPRxString_Reply
);
END_ACTION

ACTION Send_Sequence:

rTrigSendCommand(CLK := bSendCommand);

IF rTrigSendCommand.Q  THEN	
	IF stRequestCommand <> 0 THEN
		eRequestCommand	:= stRequestCommand;
	END_IF	
END_IF

// ------------------- SEND command --------------//
fbTCPSend(
	sSrvNetId	:= '',
	hSocket		:= fbTCPortCtrl_Send.hSocket,
	cbLen		:= TO_UDINT(LEN(strTCPCommand)),
	pSrc		:= ADR(strTCPCommand),
	bExecute	:= fbTCPSend.cbLen > 0 AND fbTCPSend.bBusy = FALSE,
	tTimeout	:= T#1S
);
	
	(* send data complete *)
fTrigTCPSendDone(CLK := fbTCPSend.bBusy);
IF fTrigTCPSendDone.Q = TRUE THEN

	IF fbTCPSend.bError = TRUE THEN
		bReInitialiseTCP := TRUE;
	END_IF

	strTCPLastCommand 	:= strTCPCommand;
	strLastReplyString	:= strReplyString;
	eRequestCommand 	:= E_TCPIP_RequescCommand.NONE;
	(* close off fbSendTCP *)
	fbTCPSend(bExecute 	:= FALSE);
	
	(* expece to receive reply after send finished *)
	bReceiveExpected	:= TRUE;
	
END_IF
// -------------------RECEIVE REPLY After command SENT --------------//
fbTCPReceiveAfterSend(
	bEnable			:= fbTCPortCtrl_Send.bConnected,
	hSocket			:= fbTCPortCtrl_Send.hSocket,
	tUpdateTime		:= T#100MS,
	strTCPRxString	:= strTCPRxStringReply
);

// Veryfi if reply to send command is correct //
rTrigDataReceived(CLK:=fbTCPReceiveAfterSend.bDataReceived);
IF rTrigDataReceived.Q THEN
	(*  veryfi valide response *)
	
	IF strLastReplyString = strTCPRxStringReply THEN
		bReplyOK := TRUE;
	ELSE		
		bReplyOK := FALSE;			
	END_IF
	
	GVL.aTCPxStringsReply[nIndexreply] 	:= strTCPRxStringReply;
	nIndexReply	 						:= nIndexReply + 1;
	strTCPRxStringReply 				:= '';
	bReceiveExpected					:= FALSE;
	
END_IF


//HeartBeat send every tHeartbeatInterval, IF heartbead doesent reply DO bReInitialiseTCP := TRUE
fbTON_TcpTimeout(
	IN	:= fbTCPortCtrl_Send.bConnected,
 	PT	:= tHeartbeatInterval
);
IF fbTON_TcpTimeout.Q AND (eRequestCommand = E_TCPIP_RequescCommand.NONE) THEN
	eRequestCommand 	:= E_TCPIP_RequescCommand.HeartbeatCheck;	
	fbTON_TcpTimeout(IN := FALSE);
END_IF
//////////////////////////// heartbeat handeling end ///////////////////////////////////////////////

CASE eRequestCommand OF
	
	E_TCPIP_RequescCommand.NONE:		
		strTCPCommand 	:= '';	
		strReplyString	:= '';		
	
	E_TCPIP_RequescCommand.GetUserCur:		
		strTCPCommand 	:= '<Get,UserCur>';	
		strReplyString	:= '<Get,UserCur,6>';	
		
	E_TCPIP_RequescCommand.WrongReply:		
		strTCPCommand 	:= '<Get,UserCur>';	
		strReplyString	:= '<Get,UserCur,2>';
	
	E_TCPIP_RequescCommand.HeartbeatCheck:		
		strTCPCommand 	:= '<Get,RunMode>';	
		strReplyString	:= '<Get,RunMode,0>';		
		
	E_TCPIP_RequescCommand.SetAquisitonModeON:
		strTCPCommand 	:= '<Set,Acq,1>';	
		strReplyString	:= '<Set,Acq,OK>';	
		
	E_TCPIP_RequescCommand.SetAquisitionModeOFF:
		strTCPCommand 	:= '<Set,Acq,0>';	
		strReplyString	:= '<Set,Acq,OK>';
	
END_CASE
END_ACTION

END_FUNCTION_BLOCK

// ---- POUs/SOFTWARE_lib/TCP FBs/FB_TCP_ClientPortCtrl.TcPOU
(* TCP port ctrl and monitoring for Client-Server devices *)
FUNCTION_BLOCK FB_TCP_ClientPortCtrl
VAR_INPUT
	bEnable				: BOOL;			(* set TRUE to enable TCP connection *)
	strRemoteIPAddr		: T_IPv4Addr;	(* IP address for remote device *)
	nRemotePortNo		: UINT;			(* port number for remote device *)
	tReconnectTime		: TIME;			(* TCP reconnect time *)
END_VAR
VAR_OUTPUT
	bConnected			: BOOL;			(* TRUE = TCP port is currently open *)
	bError				: BOOL;			(* TRUE = error occurred when opening TCP port *)
	nErrorID			: UDINT;		(* TRUE = error code *)
	hSocket				: T_HSocket;	(* TCP socket handle *)
	nSyncOffset			: DINT;			(* sync offset value to spread TCP Server access load *)
	eSocketState		: E_SocketConnectionState;	(* TCP socket state *)
END_VAR
VAR
	eTCPState			: E_TCPIP_State;
	strTargetIPAddr		: T_IPv4Addr;
	arrTargetIPAddr		: T_IPv4AddrArr;
	nTargetPortNo		: UDINT;
	fbTCPPortCtrl		: FB_ClientServerConnection;
END_VAR
(*
-------------------------------------------------------------------------------------------------
Date		Version	Author	Comments
-------------------------------------------------------------------------------------------------
30/01/2015	3.00.00	PB		No change

-------------------------------------------------------------------------------------------------
16/08/2012	1.40.02	PB		TCP status check now disabled if tStatusTime = T#0ms
							TCP status now check on rising edge of bEnable and every specified tStatusTime
							FB now re-connects properly if strRemoteIPAddr or nRemotePortNo are changed while TCP connection is active
							bError and nErrorID now linked directly to FB_ClientServerConnection, solves problem of auto-recovery due to incorrect status reporting.
26/01/2012	1.37.01	PB		Brackets added to ensure logic condition for when TCP connection can be disconnected is clear
22/11/2011	1.34.00	PB		tReconnectTime input added
17/11/2011	1.33.00	PB		Initial release

-------------------------------------------------------------------------------------------------
*)

CASE eTCPState OF

	(* TCP connetion not active *)
	E_TCPIP_IDLE:

		(* TCP connection is enabled *)
		IF bEnable = TRUE THEN

			(* target IP address and port number *)
			strTargetIPAddr := strRemoteIPAddr;
			nTargetPortNo := nRemotePortNo;

			(* convert target IP address to bytes *)
			arrTargetIPAddr := F_ScanIPv4AddrIds(strTargetIPAddr);
			nSyncOffset := arrTargetIPAddr[3] MOD 10;

			eTCPState := E_TCPIP_CONNECT;
		END_IF


	(* open TCP connection *)
	E_TCPIP_CONNECT:

		(* TCP connection not required or status check not active *)
		IF bEnable = FALSE (*OR (bConnect = FALSE AND bCheckStatus = FALSE)*) THEN

			eTCPState := E_TCPIP_DISCONNECT;

		(* TCP connect error or remote IP address or port number have changed while connection is active *)
		ELSIF fbTCPPortCtrl.bError = TRUE OR (strRemoteIPAddr <> strTargetIPAddr AND strTargetIPAddr <> '') OR (nRemotePortNo <> nTargetPortNo AND nTargetPortNo <> 0)THEN

			eTCPState := E_TCPIP_DISCONNECT;
		END_IF


	(* close TCP connection *)
	E_TCPIP_DISCONNECT:

		(* TCP port has been closed *)
		IF eSocketState = eSOCKET_DISCONNECTED THEN

			eTCPState := E_TCPIP_IDLE;
		END_IF

(* unknown state *)
ELSE

	eTCPState := E_TCPIP_IDLE;
END_CASE


(* TCP port connection ctrl *)
fbTCPPortCtrl(
	sSrvNetID	:= '',
	nMode		:= LISTEN_MODE_CLOSEALL, (*LISTEN_MODE_USEOPENED, CONNECT_MODE_ENABLEDBG, LISTEN_MODE_CLOSEALL*)
	sRemoteHost	:= strTargetIPAddr,
	nRemotePort	:= nTargetPortNo,
	bEnable		:= eTCPState = E_TCPIP_CONNECT,
	tReconnect	:= tReconnectTime,
	bError		=> bError,
	nErrID		=> ,
	hSocket		=> hSocket,
	eState		=> eSocketState
);

IF NOT  fbTCPPortCtrl.bBusy THEN
	nErrorID := fbTCPPortCtrl.nErrId;
END_IF
(* connected status *)
bConnected := eSocketState = eSOCKET_CONNECTED;

END_FUNCTION_BLOCK

// ---- POUs/StringFBs/FB_ExtractAnyString.TcPOU
// Extracts a sub-string defined by prefix and suffix 
// Works in one cycle but as FB to not use stack memore due to LongString data defined
FUNCTION_BLOCK FB_ExtractAnyString
VAR_INPUT
	//bExtractData			: BOOL;			
	nExtractChars			: UDINT;			(* if suffix is blank, number of data chars to extract *)
	sPrefix					: T_LongSTRING;	(* prefix string extended from T_MaxString to T_LongSTRING *)
	sSuffix					: T_LongSTRING;	(* suffix string extended from T_MaxString to T_LongSTRING *)
	bIgnoreCase				: BOOL;
	eExtractMode			: E_STRING_ExtrMode	:= E_STRING_ExtrMode.WITHOUTIDENT_REMIDENT;
	//bIncludeIdentifiers	: BOOL;
END_VAR
VAR_IN_OUT
	sDataString				: T_LongSTRING;	(* string to be searched *)
END_VAR
VAR_OUTPUT
	bStringFound			: BOOL;			(* TRUE = sub-string with matching prefix/suffix found *)
	sExtractedString		: T_LongSTRING;	(* extracted data *)
	nExtractedStringPos		: UDINT;			(* start pos of extracted string in strString *)
	nExtractedStringLen		: UDINT;
	nDataStringLen			: UDINT;
END_VAR
VAR
	
	//_rtExecute			: R_trig;
	
	_nExtractChars			: UDINT;
	_sPrefix				: T_LongSTRING;	(* prefix string *)
	_sSuffix				: T_LongSTRING;	(* suffix string *)
	_sDataString			: T_LongSTRING;	(* string to be searched *)
	
	_bIncludeIdentifiers	: BOOL;
	_bPurgeFullString		: BOOL;
	
	_nDataStringLen			: UDINT;
	_nPrefixLen				: UDINT;
	_nSuffixLen				: UDINT;
	
	_bPrefixFound			: BOOL;
	_bSuffixFound			: BOOL;
	
	_bPrefixIndex			: UDINT;
	_bTempSuffixIndex		: UDINT;
	_bSuffixIndex			: UDINT;
	
	_nStartDataPos			: UDINT;
	_nAbsolutDataPos		: UDINT;
	_nEndDataPos			: UDINT;
	_nExtractedDataLen		: UDINT;
	
	_nTerminatePos			: UDINT;
END_VAR

//	EXTRWITHIDENT						//extract with ident and dont purge left side string
//	EXTRWITHIDENT_PURGE					//extract with ident and purge left side string
//	EXTRWITHOUTIDENT					//extract with ident and dont purge left side string, both ident left in origin string 
//	EXTRWITHOUTIDENT_PURGE				//extract with ident and purge left side string, only sufix ident left in origin string
//	EXTRWITHOUTIDENT_REMIDENT			//extract with ident and dont purge left side string, no ident left in origin string
//	EXTRWITHOUTIDENT_REMIDENT_PURGE		//extract with ident and purge left side string, no ident left in origin string

//====================================================================================	
IF 	eExtractMode = E_STRING_ExtrMode.WITHIDENT 			OR 
	eExtractMode = E_STRING_ExtrMode.WITHIDENT_PURGE 	THEN
	
	_bIncludeIdentifiers	:= TRUE;
ELSE 
	_bIncludeIdentifiers	:= FALSE;
END_IF

IF 	eExtractMode = E_STRING_ExtrMode.WITHIDENT_PURGE 		OR 
	eExtractMode = E_STRING_ExtrMode.WITHOUTIDENT_PURGE 	OR 
	eExtractMode = E_STRING_ExtrMode.WITHOUTIDENT_REMIDENT_PURGE THEN
	
	_bPurgeFullString	:= LEN2(ADR(sDataString)) = SIZEOF(sDataString)-1;
ELSE 
	_bPurgeFullString	:= FALSE;
END_IF

//====================================================================================	

(* rising edge of bExecute *)
//_rtExecute(CLK := bExtractData);

//IF _rtExecute.Q THEN
	
//====================================================================================	
	bStringFound 		:= FALSE;
	
	_sDataString 		:= '';
	_sPrefix 			:= '';
	_sSuffix 			:= '';
	
	_bPrefixFound		:= FALSE;
	_bSuffixFound		:= FALSE;
		
	_bPrefixIndex		:= 0;
	_bSuffixIndex		:= 0;
		
	_nStartDataPos		:= 0;
	_nAbsolutDataPos	:= 0;
	_nEndDataPos		:= 0;
	//_ExtractedDataLen	:= 0;
	
	 (*calc string lengths *)
	_nDataStringLen 	:= LEN2(ADR(sDataString));
	_nPrefixLen 		:= LEN2(ADR(sPrefix));
	_nSuffixLen 		:= LEN2(ADR(sSuffix));
	
	_nExtractChars:= LIMIT(0, nExtractChars, _nDataStringLen);
	
	(*clear outputs*)
	nExtractedStringPos	:= 0;
	nExtractedStringLen	:= 0;
	nDataStringLen		:= _nDataStringLen;

//====================================================================================	
	
	(* matching for Prefix and Suffix is case-sesnsitive - worsk only with T_MaxString *)
	IF bIgnoreCase AND 
		_nDataStringLen < 256 	AND 
		_nPrefixLen < 256 		AND 
		_nSuffixLen < 256 		THEN
		
		(* internal comparators are all converted to lower case *)
		_sDataString 	:= F_ToLCase(sDataString);
		_sPrefix 		:= F_ToLCase(sPrefix);
		_sSuffix 		:= F_ToLCase(sSuffix);
		
	ELSE
		(* internal comparators are not changed *)
		_sDataString 	:= sDataString;
		_sPrefix 		:= sPrefix;
		_sSuffix 		:= sSuffix;
	END_IF

//====================================================================================	

	IF _nPrefixLen = 0 AND  _nExtractChars > 0 THEN
		
		_bPrefixIndex		:= 1;
		_nStartDataPos		:= 1;
		nExtractedStringPos := 1;
		
	ELSIF _nPrefixLen > 0 THEN		//if _nPrefixLen = 0 then _bPrefixIndex and _StartDataPos remains 0 from init state
		
		_bPrefixIndex	:= FIND2(ADR(_sDataString), ADR(_sPrefix));		//find search only if prefix declared on the input
	
		IF _bPrefixIndex > 0 THEN		//_bPrefixIndex as result form find can be onlu positive range
			
			_bPrefixFound := TRUE;		// _bPrefixFound guarantee _StartDataPos > 0
			_nStartDataPos 	:= SEL(_bIncludeIdentifiers, _bPrefixIndex + _nPrefixLen, _bPrefixIndex);
			_nAbsolutDataPos	:= _bPrefixIndex + _nPrefixLen;
			
			nExtractedStringPos := _nStartDataPos;
		END_IF
	END_IF	
	
//====================================================================================		

	IF _nSuffixLen = 0 AND  _nExtractChars > 0 THEN //IF only nExtractChars is declared THEN _EndDataPos pointing on elemnt determinated by nExtractChars or on last elemnt OF DataString
		
		_bSuffixIndex := _bPrefixIndex + _nPrefixLen + _nExtractChars;
		_nEndDataPos := MIN(_bSuffixIndex, _nDataStringLen);
		
		IF _nEndDataPos > _nStartDataPos THEN  // check if both pointers not point on last DataString elemnt
			_bSuffixFound := TRUE;	// _bSuffixFound guarantee _EndDataPos > 0 and found after _StartDataPos
		END_IF
		
	ELSIF _nSuffixLen > 0 THEN // if _nSuffixLen declared, then ignor nExtractChars and search for find sufix position using 
		
		// Include Sufix change shift if onle Prfix was found >> SEL(_bPrefixFound, 0, _StartDataPos - 1)
		_bTempSuffixIndex	:= FIND2(ADR(_sDataString) + SEL(_bPrefixFound, 0, _nAbsolutDataPos - 1), ADR(_sSuffix)); //find search only if sufix declared on the input and on index after prefix
		IF _bTempSuffixIndex > 0 THEN
			_bSuffixIndex	:= _bTempSuffixIndex + SEL(_bPrefixFound, 0, _nAbsolutDataPos - 1);	//Recalculate Sufix real position if sufix found or _bSuffixIndex remain 0 form init
		END_IF
		
		(*_bTempSuffixIndex gurantee that sufix was search after prefix position so _EndDataPos always greater than _StartDataPos *) 
		IF _bSuffixIndex > 0 THEN
			_bSuffixFound := TRUE;	// _bSuffixFound guarantee _EndDataPos > 0
			_nEndDataPos := SEL(_bIncludeIdentifiers,_bSuffixIndex, _bSuffixIndex + _nSuffixLen);
		END_IF
	END_IF
	
//====================================================================================		
	
	MEMSET(ADR(sExtractedString), 16#00, SIZEOF(sExtractedString));	//Clean sExtractedString area for new data

	IF _bPrefixFound AND _bSuffixFound THEN

		DELETE2(ADR(sDataString), ADR(sExtractedString), SIZEOF(sExtractedString), 
											SIZEOF(sExtractedString) - _nEndDataPos , _nEndDataPos);
		DELETE2(ADR(sExtractedString), ADR(sExtractedString), SIZEOF(sExtractedString), _nStartDataPos -1, 1);
		
	ELSIF _nPrefixLen = 0 AND _nSuffixLen = 0 AND _nExtractChars >= _nEndDataPos THEN		
		
		sExtractedString := sDataString;
		
	ELSIF _nPrefixLen = 0 AND _bSuffixFound THEN		// TO BE CONSIDERED IF WE WANT THIS CONDITION - IT WORKS LIKE LEFT
		
		_nStartDataPos := 1;
		DELETE2(ADR(sDataString), ADR(sExtractedString), SIZEOF(sExtractedString), 
										SIZEOF(sExtractedString) - _nEndDataPos , _nEndDataPos);
										
	ELSIF _bPrefixFound AND _nSuffixLen = 0 AND _nExtractChars = 0 THEN
		
		_nEndDataPos		:= _nDataStringLen;
		DELETE2(ADR(sDataString), ADR(sExtractedString), SIZEOF(sExtractedString), _nStartDataPos -1, 1);
		
	END_IF
		
	nExtractedStringLen	:= LEN2(ADR(sExtractedString));
	IF nExtractedStringLen <> 0 THEN  bStringFound := TRUE; END_IF
	
//====================================================================================
	IF NOT bStringFound AND _bPurgeFullString THEN
		
		sDataString := '';
		nDataStringLen := 0;
		
	ELSIF sExtractedString = sDataString THEN
		
		sDataString := '';
		nDataStringLen := 0;
		
	ELSIF bStringFound THEN //Terminate DataString only if endpositin for sufix is determinated and guratnee _EndDataPos greater then 0
		
		CASE eExtractMode OF

			E_STRING_ExtrMode.WITHIDENT:
			
				DELETE2(ADR(sDataString), ADR(sDataString), SIZEOF(sDataString), nExtractedStringLen, _nStartDataPos);		
					
			E_STRING_ExtrMode.WITHIDENT_PURGE:	
			
				IF _nEndDataPos = _nDataStringLen THEN
					DELETE2(ADR(sDataString), ADR(sDataString), SIZEOF(sDataString), _nEndDataPos, 1);
				ELSE
					DELETE2(ADR(sDataString), ADR(sDataString), SIZEOF(sDataString), _nEndDataPos -1, 1);
				END_IF
					
			E_STRING_ExtrMode.WITHOUTIDENT:		
			
				 DELETE2(ADR(sDataString), ADR(sDataString), SIZEOF(sDataString), nExtractedStringLen, _nStartDataPos);	
		
			E_STRING_ExtrMode.WITHOUTIDENT_PURGE:
						
				IF _nEndDataPos = _nDataStringLen THEN
					DELETE2(ADR(sDataString), ADR(sDataString), SIZEOF(sDataString), _nEndDataPos, 1);
				ELSE
					DELETE2(ADR(sDataString), ADR(sDataString), SIZEOF(sDataString), _nEndDataPos -1, 1);
				END_IF
				
			E_STRING_ExtrMode.WITHOUTIDENT_REMIDENT:
			
				DELETE2(ADR(sDataString), ADR(sDataString), SIZEOF(sDataString), 
										nExtractedStringLen + _nPrefixLen + _nSuffixLen, _bPrefixIndex);	
		
			E_STRING_ExtrMode.WITHOUTIDENT_REMIDENT_PURGE:		
						
				IF _nEndDataPos = _nDataStringLen THEN
					DELETE2(ADR(sDataString), ADR(sDataString), SIZEOF(sDataString), _nEndDataPos, 1);
				ELSE
					DELETE2(ADR(sDataString), ADR(sDataString), SIZEOF(sDataString), _bSuffixIndex + _nSuffixLen -1, 1);
				END_IF
				
		ELSE
			
			DELETE2(ADR(sDataString), ADR(sDataString), SIZEOF(sDataString), 
							nExtractedStringLen + _nPrefixLen + _nSuffixLen, _bPrefixIndex);
							
		END_CASE
	
		nDataStringLen := LEN2(ADR(sDataString));
	END_IF
//END_IF


(*

		
		IF _bSuffixIndex > _nDataStringLen THEN	//_EndDataPos cannot bi greater then _nDataStringLen due to previuse min condition
			_ExtractedDataLen := _EndDataPos -_StartDataPos + 1; // if _EndDataPos pointing on last element of sDataString, we must include it ofr extratcion
		ELSE
			_ExtractedDataLen := _EndDataPos -_StartDataPos;	//if prefix and sufix are found  _ExtractedDataLen always greater than 0
		END_IF
		
		MEMMOVE(ADR(sExtractedString),ADR(sDataString) + _StartDataPos -1 , _ExtractedDataLen);	// _StartDataPos -1 as initial adress has alredy value 1
		//MEMSET(ADR(sExtractedString) + _ExtractedDataLen, 16#00, _nDataStringLen - _ExtractedDataLen);
		
		
		
		//MEMMOVE(ADR(sExtractedString),ADR(sDataString), _EndDataPos);
		//MEMSET(ADR(sExtractedString) + _EndDataPos, 16#00, _nDataStringLen - _EndDataPos);
		
		
		
	
		IF _bSuffixIndex > _nDataStringLen THEN	//_EndDataPos cannot bi greater then _nDataStringLen due to previuse min condition
			_nTerminatePos := _EndDataPos;
		ELSE
			_nTerminatePos := SEL(_bIncludeIdentifiers, _EndDataPos + _nSuffixLen, _EndDataPos) -1; //sub 1 from final result as adressing of char start form pos 1
			//so if Terminate index should be 10 then _nTerminatePos must be 9 to add with initial addres of DataString
		END_IF
		
		IF _nDataStringLen > _nTerminatePos THEN	// guarantee we are not operating beyond DataString area
			MEMMOVE(ADR(sDataString), ADR(sDataString) + _nTerminatePos, _nDataStringLen - _nTerminatePos);
			MEMSET(ADR(sDataString) + _nDataStringLen - _nTerminatePos, 16#00, _nTerminatePos);
		ELSIF _nDataStringLen <= _nTerminatePos THEN
			sDataString := '';
		END_IF
			
	*)

END_FUNCTION_BLOCK

// ---- POUs/NewModel/FB_CAMERA_Omron.TcPOU
FUNCTION_BLOCK FB_CAMERA_Omron
VAR_INPUT
	bEnable							: BOOL;			(* set TRUE to enable TCP comms connection *)
	bConfigMode						: BOOL;			(* set TRUE to allow MV4x0 to be switched to CONFIG mode *)
	bReadCode						: BOOL;			(* set TRUE to read code *)
	stBrowseCtrl					: ST_CAMERA_BrowseCtrl;
	nReqProgram						: BYTE;			(* requested program to activate in MV4x0 *)
	sScannerIPAddr					: T_IPv4Addr;	(* scanner IP address *)
	nScannerPortNo					: UINT;			(* scanner port number *)
	stTriggerID						: ST_CAMERA_TriggerID;	(* trigger ID data, will be returned in sImageData to allow trigger and response to be aligned *)
	stOptions						: ST_CAMERA_Options;	(* MV configuration info *)
	tTimeout						: TIME;			(* timeout delay *)
	bDontParseAsGS1					: BOOL;
END_VAR
VAR_OUTPUT
	bDone							: BOOL;			(* TRUE = code scan complete *)
	bBusy							: BOOL;			(* TRUE = code scan in progress *)
	bError							: BOOL;			(* TRUE = code scan error *)
	bScannerReady					: BOOL;			(* TRUE = scanner port connected *)
	bdoTrigger						: BOOL;			(* TRG signal to camera *)
	nActiveProgram					: BYTE;			(* active program *)
	stOpState						: ST_CAMERA_OpState;	(* operating state values *)
	sImageStatus					: T_MaxString;				(* image status string *)
	stImageData						: ST_CAMERA_ImageData;		(* image data structure *)
	eSocketState					: E_SocketConnectionState;	(* TCP socket connection state *)
END_VAR
VAR
	eScannerType					: E_CAMERA_DeviceType;
	eState							: E_CAMERA_State;

	ftCameraEnable					: F_TRIG;
	rtReadCode						: R_TRIG;
	aTriggerID						: ARRAY[1..8] OF ST_CAMERA_TriggerID;
	
	fbTaskIndex						: GETCURTASKINDEX;
	tTaskTime						: TIME;
	tTCPFastTime					: TIME;

	fbTCPPortCtrl					: FB_TCP_ClientPortCtrl;
	bReInitialiseTCP				: BOOL;
	
	tonRequestStatus				: TON;
	fbTCPSend						: FB_SocketSend;
	sTCPCommand						: STRING(20);
	ftTCPSendDone					: F_TRIG;

	tofDataExpected					: TOF;
	fbTCPReceive					: FB_TCP_ReceiveLongString;
	sTCPRxString					: T_LongSTRING;
	aLogTCPRxString					: ARRAY[1..20] OF T_LongSTRING;
	aLogBytesRecieved				: ARRAY[1..20] OF UDINT;
	aTCPReceiveDone					: ARRAY[1..20] OF STRING(100);
	
	nSendCounter					: UDINT;
	nReceiveCounter					: UDINT;

	sImageDataRecived				: T_LongSTRING;
	aImageDataRecived				: ARRAY[1..20] OF STRING(100);
	sImageDataDebug					: T_LongSTRING;
	bImageData						: BOOL;

	nHeartbeat						: UDINT;
	bHeartbeat						: BOOL;
	sHeartbeatDebug					: STRING(100);
	
	nCurrentTrigger					: INT;
	nMaxImageBuffer					: INT;

	nResponseWithHeartbeatString	: UDINT;
	nResponseWithNoActiveTrigger	: UDINT;
	nResponseWithNoImageData		: UDINT;

	tonTCPTimeout					: TON;
	tonIOTimeout					: TON;
	tpAcquisitionTimer				: TP;

	fbExtractImageString 			: FB_ExtractAnyString;
	fbExtractHeartbeatString 		: FB_ExtractAnyString;
	fbDecodeImageData				: FB_CAMERA_OmronDecodeImage;
	fbBrowse						: FB_CAMERA_OmronBrowse;

	sNoImageDataDbgExt				: T_MaxString;
END_VAR
VAR CONSTANT
	sStatusRequest					: STRING := '<<K100?>>'; (* Status Request <<K126?>><<K100?>>*)
END_VAR

(*******************************************************************************************************************************)
(*Block init *)
(*******************************************************************************************************************************)
ftCameraEnable(CLK := bEnable);
IF ftCameraEnable.Q THEN
	sTCPRxString := ''; (* clears input buffer *)
END_IF

(* 1st pass of FB *)
IF tTaskTime = T#0ms THEN

	(* get current task index and PLC task time, clamped to 1ms *)
	fbTaskIndex();
	tTaskTime := MAX(UDINT_TO_TIME(_TaskInfo[fbTaskIndex.Index].CycleTime / 10000), T#1ms);

	(* fast TCP access time (10 * task time) when trigger is active *)
	tTCPFastTime := MIN(tTaskTime * 10, T#200ms);

	(* max number of active triggers supported *)
	nMaxImageBuffer := TO_INT(SIZEOF(aTriggerID) / SIZEOF(aTriggerID[1]));
END_IF

eScannerType := LIMIT(0,stOptions.eScannerType,cMAX_CAMERA_TYPES);

(*******************************************************************************************************************************)
(*TCP connection and Send receive sequences*)
(*******************************************************************************************************************************)

Connect();

Receive();

Send();

(*******************************************************************************************************************************)
(* Scanner ready and accept new trigger*)
(*******************************************************************************************************************************)

nActiveProgram 				:= nReqProgram;
stOpState.bCodeChangeActive := FALSE;

(* scanner ready when TCP port is connected, status byte is valid and code change is not in progress *)
bScannerReady := fbTCPPortCtrl.bConnected AND NOT stOpState.bTCPComsLockedUp AND NOT stOpState.bCodeChangeActive ;

(* - - - - - - - - - - - - - - - - - - - - - - - - - - - - - - - - - *)
(* scanner not ready *)
IF NOT bScannerReady THEN
	(* reset trigger and no of triggers active *)
	bdoTrigger := FALSE;
	nActiveProgram := 0;
	stOpState.nActiveTriggers := 0;
	MEMSET(ADR(stImageData), 16#00, SIZEOF(stImageData));
	MEMSET(ADR(aTriggerID), 16#00, SIZEOF(aTriggerID));
END_IF

(* - - - - - - - - - - - - - - - - - - - - - - - - - - - - - - - - - *)
stOpState.bAcceptTrigger := bScannerReady  AND NOT tpAcquisitionTimer.Q AND stOpState.nActiveTriggers < MIN(stOptions.nImageBuffer, nMaxImageBuffer);
(* rising edge of bReadCode *)
rtReadCode(CLK:= bReadCode);
(* new code requested, acquisition timer has elapsed and max triggers has not been reached *)
IF rtReadCode.Q AND stOpState.bAcceptTrigger THEN
	
	(* update number of active triggers and log TriggerID *)
	bdoTrigger := TRUE;
	
	stOpState.nActiveTriggers := stOpState.nActiveTriggers + 1;
	aTriggerID[stOpState.nActiveTriggers] := stTriggerID;

	//sTCPRxString := ''; (* clears input buffer *)
	//MEMSET(ADR(stImageData), 16#00, SIZEOF(stImageData));

	(* trigger image acquisition timer - seems never will rech its time limit, as one of input condition is one cycle triger *)
	tpAcquisitionTimer(
		IN	:= TRUE,
		PT	:= MAX(cACQUISITION_TIMER[eScannerType], tTaskTime));

(* strobe and trigger are both ON or no trigger required *)
ELSE
	(* reset trigger *)
	bdoTrigger := FALSE;
END_IF
(* reset image acquisition timer trigger *)
tpAcquisitionTimer(IN := FALSE);

(*******************************************************************************************************************************)
(* Process new code ricved codes*)
(*******************************************************************************************************************************)

Decode();

(*******************************************************************************************************************************)
(* Camera response  timeout *)
(*******************************************************************************************************************************)
(* I/O time-out delay *)
tonIOTimeout(
	IN	:= stOpState.nActiveTriggers > 0,
	PT	:= tTimeout
);

(* I/O timeout elapsed *)
IF tonIOTimeout.Q THEN

	(* reset active triggers *)
	stOpState.nResponses		:= 0;
	stOpState.nActiveTriggers 	:= 0;
	nCurrentTrigger				:= 0;
	sTCPRxString 				:= '';
	sTCPCommand 				:= '';
	MEMSET(ADR(stImageData), 16#00, SIZEOF(stImageData));
	stImageData.stTriggerID 	:= aTriggerID[1];
	stImageData.sImageStatus	:= 'I/O Timeout';
	sImageStatus 				:= stImageData.sImageStatus;
	
	(* set outputs *)
	bDone 			:= TRUE;
	bError 			:= TRUE;
END_IF

(*******************************************************************************************************************************)
(*Update Camera Status*)
(*******************************************************************************************************************************)

(* re-initialise TCP connection if TCP Send Data fails or Heartbeat times out *)
bReInitialiseTCP := (ftTCPSendDone.Q AND fbTCPSend.bError) OR stOpState.bTCPComsLockedUp;

(* busy output active while waiting for code *)
bBusy := NOT bDone AND stOpState.nActiveTriggers > 0;

(*******************************************************************************************************************************)
(* Manage browser screen*)
(*******************************************************************************************************************************)

(* browse scanner *)
fbBrowse(
	bViewLive	:= stBrowseCtrl.bBrowseLive,
	bViewDiag	:= stBrowseCtrl.bBrowseDiag,
	sIPAddress	:= sScannerIPAddr,
);

ACTION Connect:
(* TCP Port ctrl	*******************************************************************************************************)
fbTCPPortCtrl(
	bEnable			:= bEnable  AND NOT bReInitialiseTCP ,
	strRemoteIPAddr	:= sScannerIPAddr,
	nRemotePortNo	:= nScannerPortNo,
	tReconnectTime	:= T#20s,
	eSocketState	=> eSocketState
);
bReInitialiseTCP := FALSE;

IF fbTCPPortCtrl.bConnected THEN
	stOpState.nStatusByte.1 := TRUE;
	
	(* scanner in CONFIG mode *)
	IF bScannerReady = FALSE THEN

		(* clear output data *)
		nActiveProgram := 1;
		sImageStatus := '';
		MEMSET(ADR(stImageData), 16#00, SIZEOF(stImageData));
	END_IF
ELSE
	(* reset outputs *)
	sTCPCommand 				:= '';
	stOpState.nStatusByte 		:= 0;
	stOpState.nErrorCode 		:= 0;
	stOpState.bTCPComsLockedUp 	:= FALSE;
	stOpState.nActiveTriggers 	:= 0;
	nCurrentTrigger				:= 0;
	nActiveProgram 				:= 0;
	sImageStatus 				:= '';
	MEMSET(ADR(stImageData), 16#00, SIZEOF(stImageData));
END_IF


(* TCP timeout *******************************************************************************************************)
tonTCPTimeout(
	IN	:= fbTCPPortCtrl.bConnected AND stOpState.nActiveTriggers = 0 AND NOT bHeartbeat,
	PT	:= T#10s,
);

(* TCP timeout has elapsed*)
IF tonTCPTimeout.Q THEN
	(* reset TCP connection and heartbeat counter *)
	nHeartbeat 					:= 0;
	stOpState.nStatusByte.2		:= FALSE;
	stOpState.bTCPComsLockedUp 	:= TRUE;
	stOpState.nErrorCode 		:= 100;
END_IF
END_ACTION

ACTION Decode:
(* data handling sequence *)
CASE eState OF
	(* idle *)
	E_CAMERA_State.IDLE:
(* - - - - - - - - - - - - - - - - - - - - - - - - - - - - - - - - - *)
		(* further scan response expected or FB is idle *)
		IF stOpState.nActiveTriggers > 0 OR (stOpState.nActiveTriggers = 0 AND NOT bReadCode) THEN

			(* reset outputs *)
			nCurrentTrigger			:= 0;
			stOpState.nResponses	:= 0;
			
			bDone 					:= FALSE;
			bError 					:= FALSE;
			sImageStatus 			:= '';
		END_IF
	
		(* - - - - - - - - - - - - - - - - - - - - - - - - - - - - - - - - - *)	
		(* Move to wait for string to extract to complete new code recive *)	
		IF stOpState.nActiveTriggers > 0 AND stOpState.nStatusByte.2 THEN
			eState := E_CAMERA_State.IMAGE;
		END_IF
		
		(* - - - - - - - - - - - - - - - - - - - - - - - - - - - - - - - - - *)
		(* tonRequestStatus complete for heartbeat check*)
		IF stOpState.nActiveTriggers = 0 	AND
			sTCPCommand = sStatusRequest 	AND 
			stOpState.nStatusByte.1 		THEN
			
			bHeartbeat 	:= FALSE;
			sTCPCommand := '';
			eState 		:= E_CAMERA_State.HEARTBEAT;
		END_IF
		(* - - - - - - - - - - - - - - - - - - - - - - - - - - - - - - - - - *)

	(* image response *)
	E_CAMERA_State.IMAGE:

		fbExtractImageString(
			nExtractChars		:= 0, 
			sPrefix				:='$01', 
			sSuffix				:= '$04', 
			bIgnoreCase			:= FALSE, 
			eExtractMode 		:= E_STRING_ExtrMode.WITHOUTIDENT_REMIDENT_PURGE, 
			sDataString			:= sTCPRxString, 
			bStringFound		=> bImageData, 
			sExtractedString	=>, 
			nExtractedStringPos	=>,
			nExtractedStringLen	=>,
			nDataStringLen		=> 
		);
		IF fbExtractImageString.bStringFound  AND FIND2(ADR(fbExtractImageString.sExtractedString), ADR('8,0,0,1>')) <> 0  THEN
			
			nResponseWithHeartbeatString	:= nResponseWithHeartbeatString + 1;
			
		(* image response found, scanner is READY state and 1 or more triggers are active *)
		ELSIF fbExtractImageString.bStringFound  AND bScannerReady AND stOpState.nActiveTriggers > 0 THEN

			(* 1st response for current trigger *)
			IF stOpState.nResponses = 0   THEN
				(* clear sImageData *)
				nCurrentTrigger := stOpState.nActiveTriggers; 
				MEMSET(ADR(stImageData), 16#00, SIZEOF(stImageData));
			END_IF

			(* log image response string and update number of response message received *)
			sImageDataRecived := fbExtractImageString.sExtractedString;
			stOpState.nResponses := stOpState.nResponses + 1;
		
			MEMMOVE(ADR(aImageDataRecived[2]), ADR(aImageDataRecived[1]), SIZEOF(aImageDataRecived)-SIZEOF(aImageDataRecived[1]));
			aImageDataRecived[1] := F_CONCAT3(sImageDataRecived,'_', INT_TO_STRING(nCurrentTrigger));
			sImageDataDebug := sImageDataRecived;

			eState := E_CAMERA_State.DECODE;
	
		ELSIF fbExtractImageString.bStringFound AND stOpState.nActiveTriggers = 0 THEN
			
			nResponseWithNoActiveTrigger	:= nResponseWithNoActiveTrigger + 1;
			eState := E_CAMERA_State.IDLE;
			
		ELSIF tonIOTimeout.Q THEN
			
			nResponseWithNoImageData	:= nResponseWithNoImageData + 1;
			eState := E_CAMERA_State.IDLE;
		END_IF

	(* decode image data from MV4x0 *)
	E_CAMERA_State.DECODE:

		(* decode message received from scanner *)
		fbDecodeImageData(
			bExecute			:= TRUE,
			stTriggerID			:= stTriggerID,
			bDontParseAsGS1 	:= bDontParseAsGS1,
			sImageDataRecived	:= sImageDataRecived 
		);

		(* image response message received *)
		IF fbDecodeImageData.bDone = TRUE THEN

			(* image response message received *)
			IF fbDecodeImageData.bError = FALSE THEN

				(* move data to sImageData *)
				MEMMOVE(ADR(stImageData.aCodeData[stImageData.nCodesRead + 1]), ADR(fbDecodeImageData.stImageData.aCodeData[1]), SIZEOF(stImageData.aCodeData[1]) * F_SafeTo_UDINT(fbDecodeImageData.stImageData.nCodesRead));
				stImageData.nCodesRead := stImageData.nCodesRead + fbDecodeImageData.stImageData.nCodesRead;
				stImageData.tScanTime := fbDecodeImageData.stImageData.tScanTime;
			END_IF

			(* clear response data and flag *)
			sImageDataRecived := '';
			
			(* - - - - - - - - - - - - - - - - - - - - - - - - - - - - - - - - - *)
			(* ProgStandard mode and 1 response received OR ProgSequencemode and all response messages received *)
			IF (stOptions.nExpectedResp = 0 AND stOpState.nResponses = 1) 						OR 
				(stOptions.nExpectedResp > 0 AND stOpState.nResponses = stOptions.nExpectedResp) 	THEN

				(* return index for response *)
				stImageData.stTriggerID := aTriggerID[1];

				(* update trigger index array *)
				MEMMOVE(ADR(aTriggerID[1]), ADR(aTriggerID[2]), SIZEOF(aTriggerID) - SIZEOF(aTriggerID[1]));
				MEMSET(ADR(aTriggerID[nMaxImageBuffer]), 16#00, SIZEOF(aTriggerID[1]));
				
				(* reduce active triggers by 1 and reset responses *)
				stOpState.nActiveTriggers := MAX(stOpState.nActiveTriggers - 1, 0);
				//stOpState.nResponses		:= 0;
				
				(* image response data received, reset I/O timer *)
				tonIOTimeout(IN := FALSE);
				(* update status output *)
				bDone := TRUE;
				
				eState := E_CAMERA_State.IDLE;
			(* intermediate response for image received *)
			ELSE
				(* check for another image response message on next cycle *)
				eState := E_CAMERA_State.IMAGE;
			END_IF
			
			(* - - - - - - - - - - - - - - - - - - - - - - - - - - - - - - - - - *)
			(* 1 or more codes read *)
			IF stImageData.nCodesRead > 0 THEN
				(* update status outputs *)
				sImageStatus := CONCAT(INT_TO_STRING(stImageData.nCodesRead), ' code(s) read');
				stImageData.sImageStatus := sImageStatus;
			(* no codes read *)
			ELSE
				(* update status outputs *)
				sImageStatus := '0 code(s) read';
				stImageData.sImageStatus := sImageStatus;
			END_IF
			
			(* - - - - - - - - - - - - - - - - - - - - - - - - - - - - - - - - - *)
			(* close off fbDecodeImageData *)
			fbDecodeImageData(
				bExecute	:= FALSE,
				sImageDataRecived:= sImageDataRecived );
			(* - - - - - - - - - - - - - - - - - - - - - - - - - - - - - - - - - *)
		END_IF

	(* status response *)
	E_CAMERA_State.HEARTBEAT:

		//MEMMOVE(ADR(aHeartbeatDebug[2]), ADR(aHeartbeatDebug[1]), SIZEOF(aHeartbeatDebug)-SIZEOF(aHeartbeatDebug[1]));
		//aHeartbeatDebug[1] := F_CONCAT5(sTCPRxString,'_', UDINT_TO_STRING(nHeartbeat),'_', UDINT_TO_STRING(nSendCounter));
		

		(* check for status message with $04 (EOT) terminating char *)
		fbExtractHeartbeatString(
			nExtractChars		:= 0 , 
			sPrefix				:='$01', 
			sSuffix				:= '$04', 
			bIgnoreCase			:= FALSE, 
			eExtractMode 		:= E_STRING_ExtrMode.WITHOUTIDENT_REMIDENT_PURGE, 
			sDataString			:= sTCPRxString, 
			bStringFound		=> bHeartbeat, 
			sExtractedString	=>, 
			nExtractedStringPos	=> ,
			nExtractedStringLen	=> ,
			nDataStringLen		=> 
		);
		
		(* string found and response expected *)
		IF fbExtractHeartbeatString.bStringFound OR fbExtractHeartbeatString.nDataStringLen > 800 THEN
		
			stOpState.nStatusByte.2 := TRUE;
			(* update heartbeat counter *)
			nHeartbeat := nHeartbeat + 1;
			
			IF nHeartbeat = 0 OR nHeartbeat > 32000 THEN
				nHeartbeat := 1;
			END_IF
			
			sHeartbeatDebug	:= F_CONCAT5(fbExtractHeartbeatString.sExtractedString,'_', UDINT_TO_STRING(nHeartbeat),'_', UDINT_TO_STRING(nSendCounter));
			sNoImageDataDbgExt	:= sTCPRxString; 
			
			eState := E_CAMERA_State.IDLE;
			
		ELSIF tonRequestStatus.Q OR stOpState.nActiveTriggers > 0 THEN
			
			eState := E_CAMERA_State.IDLE;
			
		END_IF
(* unknown state *)
ELSE
	(* clear vars *)
	sImageStatus 				:= '';
	nCurrentTrigger				:= 0;
	stOpState.nActiveTriggers 	:= 0;
	stOpState.nResponses		:= 0;
	bdoTrigger 					:= FALSE;

	bDone 						:= FALSE;
	bError 						:= FALSE;

	eState := E_CAMERA_State.IDLE;
END_CASE
END_ACTION

ACTION Receive:
(********************************************************************************************************************************************)
(* Receive data *)
(********************************************************************************************************************************************)

tofDataExpected(IN := stOpState.nActiveTriggers > 0 OR  sTCPCommand <> '', PT:=  T#100MS);

(* poll TCP port, use tTCPFastTime when a code is expected, otherwise 200ms *)
fbTCPReceive(
	bEnable			:= fbTCPPortCtrl.bConnected,
	hSocket			:= fbTCPPortCtrl.hSocket,
	tUpdateTime		:= SEL(tofDataExpected.Q, T#200MS, tTCPFastTime),
	nSyncOffset		:= fbTCPPortCtrl.nSyncOffset * TIME_TO_DINT(tTaskTime),
	strTCPRxString	:= sTCPRxString
);

(* - - - - - - - - - - - - - - - - - - - - - - - - - - - - - - - - - *)
(* fbTCPReceive update complete for new code recive *)
IF fbTCPReceive.bDone THEN
	
	nReceiveCounter := nReceiveCounter + 1;
	MEMMOVE(ADR(aTCPReceiveDone[2]), ADR(aTCPReceiveDone[1]), SIZEOF(aTCPReceiveDone)-SIZEOF(aTCPReceiveDone[1]));
	aTCPReceiveDone[1] := F_CONCAT5(sTCPRxString,'_', UDINT_TO_STRING(nHeartbeat),'_', UDINT_TO_STRING(nReceiveCounter));
END_IF	
(* - - - - - - - - - - - - - - - - - - - - - - - - - - - - - - - - - *)
IF sTCPRxString <> '' AND sTCPRxString <> aLogTCPRxString[1] THEN
	
	MEMMOVE(ADR(aLogTCPRxString[2]) , ADR(aLogTCPRxString[1]), SIZEOF(aLogTCPRxString)-SIZEOF(aLogTCPRxString[1]));
	MEMMOVE(ADR(aLogBytesRecieved[2]) , ADR(aLogBytesRecieved[1]), SIZEOF(aLogBytesRecieved)-SIZEOF(aLogBytesRecieved[1]));
	aLogTCPRxString[1]		:= sTCPRxString;
	aLogBytesRecieved[1] 	:= fbTCPReceive.fbTCPReceive.nRecBytes;
END_IF
END_ACTION

ACTION Send:
(********************************************************************************************************************************************)
(* Send data *)
(********************************************************************************************************************************************)
tonRequestStatus(IN := stOpState.nActiveTriggers = 0 AND sTCPCommand = '' AND NOT fbTCPSend.bBusy, PT := T#5S);

IF tonRequestStatus.Q THEN
	(* request status from the camera *)
	sTCPCommand := sStatusRequest;
	
END_IF

(* access to TCPServer uses significant resource on CX1020, so TCPSend is synced with TCPReceive and ImageDecode to prevent uP task spikes *)
(* send data to TCP port *)
fbTCPSend(
	sSrvNetId	:= '',
	hSocket		:= fbTCPPortCtrl.hSocket,
	cbLen		:= LEN2(ADR(sTCPCommand)),
	pSrc		:= ADR(sTCPCommand),
	bExecute	:= tonRequestStatus.Q AND fbTCPPortCtrl.bConnected,
	//bExecute	:= fbTCPSend.cbLen > 0 AND fbTCPReceive.bDone,
	tTimeout	:= T#1s
);

IF fbTCPSend.bExecute	THEN
	nSendCounter	:= nSendCounter + 1;
END_IF

(* send data complete *)
ftTCPSendDone(CLK := fbTCPSend.bBusy);

(* TCP send complete *)
//IF ftTCPSendDone.Q OR NOT fbTCPPortCtrl.bConnected THEN
	(* clear strTCPCommand *)
//	sTCPCommand := '';
	(* close off fbSendTCPData *)
//	fbTCPSend(bExecute := FALSE);
//END_IF
END_ACTION

END_FUNCTION_BLOCK

// ---- POUs/NewModel/FB_CAMERA_HIKROBOT.TcPOU
FUNCTION_BLOCK FB_CAMERA_HIKROBOT
VAR_INPUT
	bEnable							: BOOL;			(* set TRUE to enable TCP comms connection *)
	bConfigMode						: BOOL;			(* set TRUE to allow MV4x0 to be switched to CONFIG mode *)
	bReadCode						: BOOL;			(* set TRUE to read code *)
	stBrowseCtrl					: ST_CAMERA_BrowseCtrl;
	nReqProgram						: BYTE;			(* requested program to activate in MV4x0 *)
	sScannerIPAddr					: T_IPv4Addr;	(* scanner IP address *)
	nScannerPortNo					: UINT;			(* scanner port number *)
	stTriggerID						: ST_CAMERA_TriggerID;	(* trigger ID data, will be returned in sImageData to allow trigger and response to be aligned *)
	stOptions						: ST_CAMERA_Options;	(* MV configuration info *)
	tTimeout						: TIME;			(* timeout delay *)
	bDontParseAsGS1					: BOOL;
END_VAR
VAR_OUTPUT
	bDone							: BOOL;			(* TRUE = code scan complete *)
	bBusy							: BOOL;			(* TRUE = code scan in progress *)
	bError							: BOOL;			(* TRUE = code scan error *)
	bScannerReady					: BOOL;			(* TRUE = scanner port connected *)
	bdoTrigger						: BOOL;			(* TRG signal to camera *)
	nActiveProgram					: BYTE;			(* active program *)
	stOpState						: ST_CAMERA_OpState;	(* operating state values *)
	sImageStatus					: T_MaxString;				(* image status string *)
	stImageData						: ST_CAMERA_ImageData;		(* image data structure *)
	eSocketState					: E_SocketConnectionState;	(* TCP socket connection state *)
END_VAR
VAR
	eScannerType					: E_CAMERA_DeviceType;
	eState							: E_CAMERA_State;

	ftCameraEnable					: F_TRIG;
	rtReadCode						: R_TRIG;
	aTriggerID						: ARRAY[1..8] OF ST_CAMERA_TriggerID;
	
	fbTaskIndex						: GETCURTASKINDEX;
	tTaskTime						: TIME;
	tTCPFastTime					: TIME;

	fbTCPPortCtrl					: FB_TCP_ClientPortCtrl;
	bReInitialiseTCP				: BOOL;
	
	tonRequestStatus				: TON;
	fbTCPSend						: FB_SocketSend;
	sTCPCommand						: STRING(20);
	ftTCPSendDone					: F_TRIG;

	tofDataExpected					: TOF;
	fbTCPReceive					: FB_TCP_ReceiveLongString;
	sTCPRxString					: T_LongSTRING;
	aLogTCPRxString					: ARRAY[1..20] OF T_LongSTRING;
	aLogBytesRecieved				: ARRAY[1..20] OF UDINT;
	aTCPReceiveDone					: ARRAY[1..20] OF STRING(100);
	
	nSendCounter					: UDINT;
	nReceiveCounter					: UDINT;

	sImageDataRecived				: T_LongSTRING;
	aImageDataRecived				: ARRAY[1..20] OF STRING(100);
	sImageDataDebug					: T_LongSTRING;
	bImageData						: BOOL;

	nHeartbeat						: UDINT;
	bHeartbeat						: BOOL;
	sHeartbeatDebug					: STRING(100);
	
	nCurrentTrigger					: INT;
	nMaxImageBuffer					: INT;

	nResponseWithHeartbeatString	: UDINT;
	nResponseWithNoActiveTrigger	: UDINT;
	nResponseWithNoImageData		: UDINT;

	tonTCPTimeout					: TON;
	tonIOTimeout					: TON;
	tpAcquisitionTimer				: TP;

	fbExtractImageString 			: FB_ExtractAnyString;
	fbExtractHeartbeatString 		: FB_ExtractAnyString;
	fbDecodeImageData				: FB_CAMERA_OmronDecodeImage;
	fbBrowse						: FB_CAMERA_OmronBrowse;

	sNoImageDataDbgExt				: T_MaxString;
END_VAR
VAR CONSTANT
	sStatusRequest					: STRING := '<<K100?>>'; (* Status Request <<K126?>><<K100?>>*)
END_VAR

(*******************************************************************************************************************************)
(*Block init *)
(*******************************************************************************************************************************)
ftCameraEnable(CLK := bEnable);
IF ftCameraEnable.Q THEN
	sTCPRxString := ''; (* clears input buffer *)
END_IF

(* 1st pass of FB *)
IF tTaskTime = T#0ms THEN

	(* get current task index and PLC task time, clamped to 1ms *)
	fbTaskIndex();
	tTaskTime := MAX(UDINT_TO_TIME(_TaskInfo[fbTaskIndex.Index].CycleTime / 10000), T#1ms);

	(* fast TCP access time (10 * task time) when trigger is active *)
	tTCPFastTime := MIN(tTaskTime * 10, T#200ms);

	(* max number of active triggers supported *)
	nMaxImageBuffer := TO_INT(SIZEOF(aTriggerID) / SIZEOF(aTriggerID[1]));
END_IF

eScannerType := LIMIT(0,stOptions.eScannerType,cMAX_CAMERA_TYPES);

(*******************************************************************************************************************************)
(*TCP connection and Send receive sequences*)
(*******************************************************************************************************************************)

Connect();

Receive();

Send();

(*******************************************************************************************************************************)
(* Scanner ready and accept new trigger*)
(*******************************************************************************************************************************)

nActiveProgram 				:= nReqProgram;
stOpState.bCodeChangeActive := FALSE;

(* scanner ready when TCP port is connected, status byte is valid and code change is not in progress *)
bScannerReady := fbTCPPortCtrl.bConnected AND NOT stOpState.bTCPComsLockedUp AND NOT stOpState.bCodeChangeActive ;

(* - - - - - - - - - - - - - - - - - - - - - - - - - - - - - - - - - *)
(* scanner not ready *)
IF NOT bScannerReady THEN
	(* reset trigger and no of triggers active *)
	bdoTrigger := FALSE;
	nActiveProgram := 0;
	stOpState.nActiveTriggers := 0;
	MEMSET(ADR(stImageData), 16#00, SIZEOF(stImageData));
	MEMSET(ADR(aTriggerID), 16#00, SIZEOF(aTriggerID));
END_IF

(* - - - - - - - - - - - - - - - - - - - - - - - - - - - - - - - - - *)
stOpState.bAcceptTrigger := bScannerReady  AND NOT tpAcquisitionTimer.Q AND stOpState.nActiveTriggers < MIN(stOptions.nImageBuffer, nMaxImageBuffer);
(* rising edge of bReadCode *)
rtReadCode(CLK:= bReadCode);
(* new code requested, acquisition timer has elapsed and max triggers has not been reached *)
IF rtReadCode.Q AND stOpState.bAcceptTrigger THEN
	
	(* update number of active triggers and log TriggerID *)
	bdoTrigger := TRUE;
	
	stOpState.nActiveTriggers := stOpState.nActiveTriggers + 1;
	aTriggerID[stOpState.nActiveTriggers] := stTriggerID;

	//sTCPRxString := ''; (* clears input buffer *)
	//MEMSET(ADR(stImageData), 16#00, SIZEOF(stImageData));

	(* trigger image acquisition timer - seems never will rech its time limit, as one of input condition is one cycle triger *)
	tpAcquisitionTimer(
		IN	:= TRUE,
		PT	:= MAX(cACQUISITION_TIMER[eScannerType], tTaskTime));

(* strobe and trigger are both ON or no trigger required *)
ELSE
	(* reset trigger *)
	bdoTrigger := FALSE;
END_IF
(* reset image acquisition timer trigger *)
tpAcquisitionTimer(IN := FALSE);

(*******************************************************************************************************************************)
(* Process new code ricved codes*)
(*******************************************************************************************************************************)

Decode();

(*******************************************************************************************************************************)
(* Camera response  timeout *)
(*******************************************************************************************************************************)
(* I/O time-out delay *)
tonIOTimeout(
	IN	:= stOpState.nActiveTriggers > 0,
	PT	:= tTimeout
);

(* I/O timeout elapsed *)
IF tonIOTimeout.Q THEN

	(* reset active triggers *)
	stOpState.nResponses		:= 0;
	stOpState.nActiveTriggers 	:= 0;
	nCurrentTrigger				:= 0;
	sTCPRxString 				:= '';
	sTCPCommand 				:= '';
	MEMSET(ADR(stImageData), 16#00, SIZEOF(stImageData));
	stImageData.stTriggerID 	:= aTriggerID[1];
	stImageData.sImageStatus	:= 'I/O Timeout';
	sImageStatus 				:= stImageData.sImageStatus;
	
	(* set outputs *)
	bDone 			:= TRUE;
	bError 			:= TRUE;
END_IF

(*******************************************************************************************************************************)
(*Update Camera Status*)
(*******************************************************************************************************************************)

(* re-initialise TCP connection if TCP Send Data fails or Heartbeat times out *)
bReInitialiseTCP := (ftTCPSendDone.Q AND fbTCPSend.bError) OR stOpState.bTCPComsLockedUp;

(* busy output active while waiting for code *)
bBusy := NOT bDone AND stOpState.nActiveTriggers > 0;

(*******************************************************************************************************************************)
(* Manage browser screen*)
(*******************************************************************************************************************************)

(* browse scanner *)
fbBrowse(
	bViewLive	:= stBrowseCtrl.bBrowseLive,
	bViewDiag	:= stBrowseCtrl.bBrowseDiag,
	sIPAddress	:= sScannerIPAddr,
);

ACTION Connect:
(* TCP Port ctrl	*******************************************************************************************************)
fbTCPPortCtrl(
	bEnable			:= bEnable  AND NOT bReInitialiseTCP ,
	strRemoteIPAddr	:= sScannerIPAddr,
	nRemotePortNo	:= nScannerPortNo,
	tReconnectTime	:= T#20s,
	eSocketState	=> eSocketState
);
bReInitialiseTCP := FALSE;

IF fbTCPPortCtrl.bConnected THEN
	stOpState.nStatusByte.1 := TRUE;
	
	(* scanner in CONFIG mode *)
	IF bScannerReady = FALSE THEN

		(* clear output data *)
		nActiveProgram := 1;
		sImageStatus := '';
		MEMSET(ADR(stImageData), 16#00, SIZEOF(stImageData));
	END_IF
ELSE
	(* reset outputs *)
	sTCPCommand 				:= '';
	stOpState.nStatusByte 		:= 0;
	stOpState.nErrorCode 		:= 0;
	stOpState.bTCPComsLockedUp 	:= FALSE;
	stOpState.nActiveTriggers 	:= 0;
	nCurrentTrigger				:= 0;
	nActiveProgram 				:= 0;
	sImageStatus 				:= '';
	MEMSET(ADR(stImageData), 16#00, SIZEOF(stImageData));
END_IF


(* TCP timeout *******************************************************************************************************)
tonTCPTimeout(
	IN	:= fbTCPPortCtrl.bConnected AND stOpState.nActiveTriggers = 0 AND NOT bHeartbeat,
	PT	:= T#10s,
);

(* TCP timeout has elapsed*)
IF tonTCPTimeout.Q THEN
	(* reset TCP connection and heartbeat counter *)
	nHeartbeat 					:= 0;
	stOpState.nStatusByte.2		:= FALSE;
	stOpState.bTCPComsLockedUp 	:= TRUE;
	stOpState.nErrorCode 		:= 100;
END_IF
END_ACTION

ACTION Decode:
(* data handling sequence *)
CASE eState OF
	(* idle *)
	E_CAMERA_State.IDLE:
(* - - - - - - - - - - - - - - - - - - - - - - - - - - - - - - - - - *)
		(* further scan response expected or FB is idle *)
		IF stOpState.nActiveTriggers > 0 OR (stOpState.nActiveTriggers = 0 AND NOT bReadCode) THEN

			(* reset outputs *)
			nCurrentTrigger			:= 0;
			stOpState.nResponses	:= 0;
			
			bDone 					:= FALSE;
			bError 					:= FALSE;
			sImageStatus 			:= '';
		END_IF
	
		(* - - - - - - - - - - - - - - - - - - - - - - - - - - - - - - - - - *)	
		(* Move to wait for string to extract to complete new code recive *)	
		IF stOpState.nActiveTriggers > 0 AND stOpState.nStatusByte.2 THEN
			eState := E_CAMERA_State.IMAGE;
		END_IF
		
		(* - - - - - - - - - - - - - - - - - - - - - - - - - - - - - - - - - *)
		(* tonRequestStatus complete for heartbeat check*)
		IF stOpState.nActiveTriggers = 0 	AND
			sTCPCommand = sStatusRequest 	AND 
			stOpState.nStatusByte.1 		THEN
			
			bHeartbeat 	:= FALSE;
			sTCPCommand := '';
			eState 		:= E_CAMERA_State.HEARTBEAT;
		END_IF
		(* - - - - - - - - - - - - - - - - - - - - - - - - - - - - - - - - - *)

	(* image response *)
	E_CAMERA_State.IMAGE:

		fbExtractImageString(
			nExtractChars		:= 0, 
			sPrefix				:='$01', 
			sSuffix				:= '$04', 
			bIgnoreCase			:= FALSE, 
			eExtractMode 		:= E_STRING_ExtrMode.WITHOUTIDENT_REMIDENT_PURGE, 
			sDataString			:= sTCPRxString, 
			bStringFound		=> bImageData, 
			sExtractedString	=>, 
			nExtractedStringPos	=>,
			nExtractedStringLen	=>,
			nDataStringLen		=> 
		);
		IF fbExtractImageString.bStringFound  AND FIND2(ADR(fbExtractImageString.sExtractedString), ADR('8,0,0,1>')) <> 0  THEN
			
			nResponseWithHeartbeatString	:= nResponseWithHeartbeatString + 1;
			
		(* image response found, scanner is READY state and 1 or more triggers are active *)
		ELSIF fbExtractImageString.bStringFound  AND bScannerReady AND stOpState.nActiveTriggers > 0 THEN

			(* 1st response for current trigger *)
			IF stOpState.nResponses = 0   THEN
				(* clear sImageData *)
				nCurrentTrigger := stOpState.nActiveTriggers; 
				MEMSET(ADR(stImageData), 16#00, SIZEOF(stImageData));
			END_IF

			(* log image response string and update number of response message received *)
			sImageDataRecived := fbExtractImageString.sExtractedString;
			stOpState.nResponses := stOpState.nResponses + 1;
		
			MEMMOVE(ADR(aImageDataRecived[2]), ADR(aImageDataRecived[1]), SIZEOF(aImageDataRecived)-SIZEOF(aImageDataRecived[1]));
			aImageDataRecived[1] := F_CONCAT3(sImageDataRecived,'_', INT_TO_STRING(nCurrentTrigger));
			sImageDataDebug := sImageDataRecived;

			eState := E_CAMERA_State.DECODE;
	
		ELSIF fbExtractImageString.bStringFound AND stOpState.nActiveTriggers = 0 THEN
			
			nResponseWithNoActiveTrigger	:= nResponseWithNoActiveTrigger + 1;
			eState := E_CAMERA_State.IDLE;
			
		ELSIF tonIOTimeout.Q THEN
			
			nResponseWithNoImageData	:= nResponseWithNoImageData + 1;
			eState := E_CAMERA_State.IDLE;
		END_IF

	(* decode image data from MV4x0 *)
	E_CAMERA_State.DECODE:

		(* decode message received from scanner *)
		fbDecodeImageData(
			bExecute			:= TRUE,
			stTriggerID			:= stTriggerID,
			bDontParseAsGS1 	:= bDontParseAsGS1,
			sImageDataRecived	:= sImageDataRecived 
		);

		(* image response message received *)
		IF fbDecodeImageData.bDone = TRUE THEN

			(* image response message received *)
			IF fbDecodeImageData.bError = FALSE THEN

				(* move data to sImageData *)
				MEMMOVE(ADR(stImageData.aCodeData[stImageData.nCodesRead + 1]), ADR(fbDecodeImageData.stImageData.aCodeData[1]), SIZEOF(stImageData.aCodeData[1]) * F_SafeTo_UDINT(fbDecodeImageData.stImageData.nCodesRead));
				stImageData.nCodesRead := stImageData.nCodesRead + fbDecodeImageData.stImageData.nCodesRead;
				stImageData.tScanTime := fbDecodeImageData.stImageData.tScanTime;
			END_IF

			(* clear response data and flag *)
			sImageDataRecived := '';
			
			(* - - - - - - - - - - - - - - - - - - - - - - - - - - - - - - - - - *)
			(* ProgStandard mode and 1 response received OR ProgSequencemode and all response messages received *)
			IF (stOptions.nExpectedResp = 0 AND stOpState.nResponses = 1) 						OR 
				(stOptions.nExpectedResp > 0 AND stOpState.nResponses = stOptions.nExpectedResp) 	THEN

				(* return index for response *)
				stImageData.stTriggerID := aTriggerID[1];

				(* update trigger index array *)
				MEMMOVE(ADR(aTriggerID[1]), ADR(aTriggerID[2]), SIZEOF(aTriggerID) - SIZEOF(aTriggerID[1]));
				MEMSET(ADR(aTriggerID[nMaxImageBuffer]), 16#00, SIZEOF(aTriggerID[1]));
				
				(* reduce active triggers by 1 and reset responses *)
				stOpState.nActiveTriggers := MAX(stOpState.nActiveTriggers - 1, 0);
				//stOpState.nResponses		:= 0;
				
				(* image response data received, reset I/O timer *)
				tonIOTimeout(IN := FALSE);
				(* update status output *)
				bDone := TRUE;
				
				eState := E_CAMERA_State.IDLE;
			(* intermediate response for image received *)
			ELSE
				(* check for another image response message on next cycle *)
				eState := E_CAMERA_State.IMAGE;
			END_IF
			
			(* - - - - - - - - - - - - - - - - - - - - - - - - - - - - - - - - - *)
			(* 1 or more codes read *)
			IF stImageData.nCodesRead > 0 THEN
				(* update status outputs *)
				sImageStatus := CONCAT(INT_TO_STRING(stImageData.nCodesRead), ' code(s) read');
				stImageData.sImageStatus := sImageStatus;
			(* no codes read *)
			ELSE
				(* update status outputs *)
				sImageStatus := '0 code(s) read';
				stImageData.sImageStatus := sImageStatus;
			END_IF
			
			(* - - - - - - - - - - - - - - - - - - - - - - - - - - - - - - - - - *)
			(* close off fbDecodeImageData *)
			fbDecodeImageData(
				bExecute	:= FALSE,
				sImageDataRecived:= sImageDataRecived );
			(* - - - - - - - - - - - - - - - - - - - - - - - - - - - - - - - - - *)
		END_IF

	(* status response *)
	E_CAMERA_State.HEARTBEAT:

		//MEMMOVE(ADR(aHeartbeatDebug[2]), ADR(aHeartbeatDebug[1]), SIZEOF(aHeartbeatDebug)-SIZEOF(aHeartbeatDebug[1]));
		//aHeartbeatDebug[1] := F_CONCAT5(sTCPRxString,'_', UDINT_TO_STRING(nHeartbeat),'_', UDINT_TO_STRING(nSendCounter));
		

		(* check for status message with $04 (EOT) terminating char *)
		fbExtractHeartbeatString(
			nExtractChars		:= 0 , 
			sPrefix				:='$01', 
			sSuffix				:= '$04', 
			bIgnoreCase			:= FALSE, 
			eExtractMode 		:= E_STRING_ExtrMode.WITHOUTIDENT_REMIDENT_PURGE, 
			sDataString			:= sTCPRxString, 
			bStringFound		=> bHeartbeat, 
			sExtractedString	=>, 
			nExtractedStringPos	=> ,
			nExtractedStringLen	=> ,
			nDataStringLen		=> 
		);
		
		(* string found and response expected *)
		IF fbExtractHeartbeatString.bStringFound OR fbExtractHeartbeatString.nDataStringLen > 800 THEN
		
			stOpState.nStatusByte.2 := TRUE;
			(* update heartbeat counter *)
			nHeartbeat := nHeartbeat + 1;
			
			IF nHeartbeat = 0 OR nHeartbeat > 32000 THEN
				nHeartbeat := 1;
			END_IF
			
			sHeartbeatDebug	:= F_CONCAT5(fbExtractHeartbeatString.sExtractedString,'_', UDINT_TO_STRING(nHeartbeat),'_', UDINT_TO_STRING(nSendCounter));
			sNoImageDataDbgExt	:= sTCPRxString; 
			
			eState := E_CAMERA_State.IDLE;
			
		ELSIF tonRequestStatus.Q OR stOpState.nActiveTriggers > 0 THEN
			
			eState := E_CAMERA_State.IDLE;
			
		END_IF
(* unknown state *)
ELSE
	(* clear vars *)
	sImageStatus 				:= '';
	nCurrentTrigger				:= 0;
	stOpState.nActiveTriggers 	:= 0;
	stOpState.nResponses		:= 0;
	bdoTrigger 					:= FALSE;

	bDone 						:= FALSE;
	bError 						:= FALSE;

	eState := E_CAMERA_State.IDLE;
END_CASE
END_ACTION

ACTION Receive:
(********************************************************************************************************************************************)
(* Receive data *)
(********************************************************************************************************************************************)

tofDataExpected(IN := stOpState.nActiveTriggers > 0 OR  sTCPCommand <> '', PT:=  T#100MS);

(* poll TCP port, use tTCPFastTime when a code is expected, otherwise 200ms *)
fbTCPReceive(
	bEnable			:= fbTCPPortCtrl.bConnected,
	hSocket			:= fbTCPPortCtrl.hSocket,
	tUpdateTime		:= SEL(tofDataExpected.Q, T#200MS, tTCPFastTime),
	nSyncOffset		:= fbTCPPortCtrl.nSyncOffset * TIME_TO_DINT(tTaskTime),
	strTCPRxString	:= sTCPRxString
);

(* - - - - - - - - - - - - - - - - - - - - - - - - - - - - - - - - - *)
(* fbTCPReceive update complete for new code recive *)
IF fbTCPReceive.bDone THEN
	
	nReceiveCounter := nReceiveCounter + 1;
	MEMMOVE(ADR(aTCPReceiveDone[2]), ADR(aTCPReceiveDone[1]), SIZEOF(aTCPReceiveDone)-SIZEOF(aTCPReceiveDone[1]));
	aTCPReceiveDone[1] := F_CONCAT5(sTCPRxString,'_', UDINT_TO_STRING(nHeartbeat),'_', UDINT_TO_STRING(nReceiveCounter));
END_IF	
(* - - - - - - - - - - - - - - - - - - - - - - - - - - - - - - - - - *)
IF sTCPRxString <> '' AND sTCPRxString <> aLogTCPRxString[1] THEN
	
	MEMMOVE(ADR(aLogTCPRxString[2]) , ADR(aLogTCPRxString[1]), SIZEOF(aLogTCPRxString)-SIZEOF(aLogTCPRxString[1]));
	MEMMOVE(ADR(aLogBytesRecieved[2]) , ADR(aLogBytesRecieved[1]), SIZEOF(aLogBytesRecieved)-SIZEOF(aLogBytesRecieved[1]));
	aLogTCPRxString[1]		:= sTCPRxString;
	aLogBytesRecieved[1] 	:= fbTCPReceive.fbTCPReceive.nRecBytes;
END_IF
END_ACTION

ACTION Send:
(********************************************************************************************************************************************)
(* Send data *)
(********************************************************************************************************************************************)
tonRequestStatus(IN := stOpState.nActiveTriggers = 0 AND sTCPCommand = '' AND NOT fbTCPSend.bBusy, PT := T#5S);

IF tonRequestStatus.Q THEN
	(* request status from the camera *)
	sTCPCommand := sStatusRequest;
	
END_IF

(* access to TCPServer uses significant resource on CX1020, so TCPSend is synced with TCPReceive and ImageDecode to prevent uP task spikes *)
(* send data to TCP port *)
fbTCPSend(
	sSrvNetId	:= '',
	hSocket		:= fbTCPPortCtrl.hSocket,
	cbLen		:= LEN2(ADR(sTCPCommand)),
	pSrc		:= ADR(sTCPCommand),
	bExecute	:= tonRequestStatus.Q AND fbTCPPortCtrl.bConnected,
	//bExecute	:= fbTCPSend.cbLen > 0 AND fbTCPReceive.bDone,
	tTimeout	:= T#1s
);

IF fbTCPSend.bExecute	THEN
	nSendCounter	:= nSendCounter + 1;
END_IF

(* send data complete *)
ftTCPSendDone(CLK := fbTCPSend.bBusy);

(* TCP send complete *)
//IF ftTCPSendDone.Q OR NOT fbTCPPortCtrl.bConnected THEN
	(* clear strTCPCommand *)
//	sTCPCommand := '';
	(* close off fbSendTCPData *)
//	fbTCPSend(bExecute := FALSE);
//END_IF
END_ACTION

END_FUNCTION_BLOCK

// ---- POUs/SOFTWARE_lib/TCP FBs/FB_TCP_ClientPortCtrl_V2.TcPOU
(* TCP port ctrl and monitoring for Client-Server devices *)
FUNCTION_BLOCK FB_TCP_ClientPortCtrl_V2
VAR_INPUT
	bEnable				: BOOL;			(* set TRUE to enable device presence monitoring *)
	bConnect			: BOOL;			(* set TRUE to open the TCP connection *)
	strRemoteIPAddr		: T_IPv4Addr;	(* remote IP address *)
	nRemotePortNo		: UDINT;		(* remote port number *)
	tReconnectTime		: TIME;			(* TCP reconnect time *)
	tStatusTime			: TIME;			(* status check time, set to T#0s to disable status checking *)
END_VAR
VAR_OUTPUT
	bConnected			: BOOL;			(* TRUE = TCP port is currently open *)
	bError				: BOOL;			(* TRUE = error occurred when opening TCP port *)
	nErrorID			: UDINT;		(* TRUE = error code *)
	bStatusOK			: BOOL;			(* TRUE = TCP port was opened successfully on last attempt *)
	hSocket				: T_HSocket;	(* TCP socket handle *)
	eSocketState		: E_SocketConnectionState;	(* TCP socket state *)
END_VAR
VAR
	strTargetIPAddr		: T_IPv4Addr;
	nTargetPortNo		: UDINT;
	fbTCPPortCtrl		: FB_ClientServerConnection;
	bStatusCheckActive	: BOOL;
	fbEnable			: R_TRIG;
	bCheckStatus		: BOOL;
	eTCPState			: E_TCPIP_State;
	fbCheckStatus		: TON;
END_VAR
(*
-------------------------------------------------------------------------------------------------
Date		Version	Author	Comments
-------------------------------------------------------------------------------------------------
16/08/2012	1.40.02	PB		TCP status check now disabled if tStatusTime = T#0ms
							TCP status now check on rising edge of bEnable and every specified tStatusTime.
							FB now re-connects properly if strRemoteIPAddr or nRemotePortNo are changed while TCP connection is active.
							bError and nErrorID now linked directly to FB_ClientServerConnection, solves problem of auto-recovery due to incorrect status reporting.
26/01/2012	1.37.01	PB		Brackets added to ensure logic condition for when TCP connection can be disconnected is clear.
22/11/2011	1.34.00	PB		tReconnectTime input added.
17/11/2011	1.33.00	PB		Initial release

-------------------------------------------------------------------------------------------------
*)

(* rising edge of bEnable *)
fbEnable(CLK := bEnable);

(* TCP status check timer *)
fbCheckStatus(
	IN	:= bEnable,
	PT	:= tStatusTime
);

(* if configured, check device status when connection is enabled and every status period *)
IF tStatusTime > T#0ms AND (fbEnable.Q = TRUE OR fbCheckStatus.Q = TRUE) THEN

	(* reset TCP status check timer *)
	fbCheckStatus(IN := FALSE);

	(* set flag to trigger next status check *)
	bCheckStatus := TRUE;
END_IF


CASE eTCPState OF

	(* TCP connetion not active *)
	E_TCPIP_IDLE:

		(* TCP connection is enabled *)
		IF bEnable = TRUE THEN

			(* TCP connection is required *)
			IF bConnect = TRUE THEN

				(* target IP address and port number *)
				strTargetIPAddr := strRemoteIPAddr;
				nTargetPortNo := nRemotePortNo;

				eTCPState := E_TCPIP_CONNECT;

			(* status check required *)
			ELSIF bCheckStatus = TRUE THEN

				(* target IP address and port number *)
				strTargetIPAddr := strRemoteIPAddr;
				nTargetPortNo := nRemotePortNo;

				(* update status check flags *)
				bCheckStatus := FALSE;
				bStatusCheckActive := TRUE;

				eTCPState := E_TCPIP_CONNECT;
			END_IF

		(* TCP connection is disabled *)
		ELSE

			bCheckStatus := FALSE;
			bStatusCheckActive := FALSE;

			(* reset outputs *)
			bConnected := FALSE;
			bStatusOK := FALSE;
			MEMSET(ADR(hSocket), 16#00, SIZEOF(hSocket));
			MEMSET(ADR(eSocketState), 16#00, SIZEOF(eSocketState));
		END_IF


	(* open TCP connection *)
	E_TCPIP_CONNECT:

		IF fbTCPPortCtrl.bBusy = FALSE THEN

			(* TCP connection not required and status check is not active *)
			IF bEnable = FALSE OR (bConnect = FALSE AND bStatusCheckActive = FALSE) THEN
	
				eTCPState := E_TCPIP_DISCONNECT;

			(* TCP connection error *)
			ELSIF fbTCPPortCtrl.bError = TRUE THEN
	
				(* update outputs *)
				bConnected := FALSE;
				bStatusOK := FALSE;

				eTCPState := E_TCPIP_DISCONNECT;
	
			(* TCP connection opened OK *)
			ELSIF eSocketState = eSOCKET_CONNECTED THEN
	
				(* status check complete *)
				bStatusCheckActive := FALSE;

				bConnected := TRUE;
				bStatusOK := TRUE;
			END_IF
		END_IF

	(* close TCP connection *)
	E_TCPIP_DISCONNECT:

		(* ensure status check is cancelled *)
		bStatusCheckActive := FALSE;

		(* reset bConnected flag *)
		bConnected := FALSE;

		(* TCP port has been closed *)
		IF eSocketState = eSOCKET_DISCONNECTED THEN

			eTCPState := E_TCPIP_IDLE;
		END_IF

	(* unknown state *)
	ELSE

		(* reset outputs *)
		bConnected := FALSE;
		bStatusOK := FALSE;
		MEMSET(ADR(hSocket), 16#00, SIZEOF(hSocket));
		MEMSET(ADR(eSocketState), 16#00, SIZEOF(eSocketState));

		eTCPState := E_TCPIP_IDLE;

END_CASE


(* remote IP address or port number have changed while connection is active *)
IF (strRemoteIPAddr <> strTargetIPAddr AND strTargetIPAddr <> '') OR (nRemotePortNo <> nTargetPortNo AND nTargetPortNo <> 0) THEN

	(* reset outputs *)
	bConnected := FALSE;
	bStatusOK := FALSE;

	eTCPState := E_TCPIP_DISCONNECT;
END_IF

(* TCP port connection ctrl *)
fbTCPPortCtrl(
	sSrvNetID	:= '',
	nMode		:= LISTEN_MODE_USEOPENED, (*CONNECT_MODE_ENABLEDBG,*)
	sRemoteHost	:= strTargetIPAddr,
	nRemotePort	:= nTargetPortNo,
	bEnable		:= eTCPState = E_TCPIP_CONNECT,
	tReconnect	:= tReconnectTime,
	bError		=> bError,
	nErrID		=> nErrorID,
	hSocket		=> hSocket,
	eState		=> eSocketState
);

END_FUNCTION_BLOCK

// ---- POUs/SOFTWARE_lib/TCP FBs/FB_TCP_CloseAllPorts.TcPOU
(* close all TCP ports, re-tries at start-up until TCP Server is running *)
FUNCTION_BLOCK FB_TCP_CloseAllPorts
VAR_INPUT
	bExecute		: BOOL;		(* set TRUE to close any TCP connections previously opened by PLC runtime *)
	tTimeout		: TIME;		(* timeout before bError is set in case TCP Server is not installed *)
END_VAR
VAR_OUTPUT
	bDone			: BOOL;		(* TRUE = close all ports complete *)
	bBusy			: BOOL;		(* TRUE = close all ports in progress *)
	bError			: BOOL;		(* TRUE = TCP server error after tTimeout *)
	nErrorID		: UDINT;	(* TCP Server error code *)
END_VAR
VAR
	fbExecute		: R_TRIG;
	eState			: E_TCPIP_State;
	nCycles			: INT;
	fbCloseAllPorts	: FB_SocketCloseAll;
	fbTimer			: TON;
END_VAR
(*
-------------------------------------------------------------------------------------------------
DATE		Version	Author	Comments
-------------------------------------------------------------------------------------------------
06/03/2015	3.05.00	PB		Initial release.

-------------------------------------------------------------------------------------------------
*)

(* rising edge of bExecute *)
fbExecute(CLK := bExecute);

CASE eState OF

	(* idle *)
	E_TCPIP_IDLE:

		(* rising edge of bExecute *)
		IF fbExecute.Q = TRUE THEN

			(* update outputs *)
			bDone := FALSE;
			bBusy := TRUE;
			bError := FALSE;
			nErrorID := 0;

			(* reset timer *)
			fbTimer(IN := FALSE);
			nCycles := 0;

			eState := E_TCPIP_CLOSEALL;

		(* bExecute has been reset *)
		ELSIF bExecute = FALSE THEN

			(* reset outputs *)
			bDone := FALSE;
			bBusy := FALSE;
			bError := FALSE;
			nErrorID := 0;
		END_IF


	(* close all TCP sockets *)
	E_TCPIP_CLOSEALL:

		(* TCP server timer *)
		fbTimer(
			IN	:= TRUE,
			PT	:= tTimeout
		);

		(* close all TCP ports for PLC runtime *)
		fbCloseAllPorts(
			sSrvNetId	:= '',
			bExecute	:= TRUE,
			tTimeout	:= T#500ms
		);

		(* command complete *)
		IF fbCloseAllPorts.bBusy = FALSE THEN

			(* update cycle counter *)
			nCycles := nCycles + 1;

			(* command completed OK *)
			IF fbCloseAllPorts.bError = FALSE THEN

				eState := E_TCPIP_DONE;

			(* command error *)
			ELSE

				(* timer has elapsed *)
				IF fbTimer.Q = TRUE THEN

					(* TCP server error *)
					bError := TRUE;
					nErrorID := fbCloseAllPorts.nErrId;

					eState := E_TCPIP_DONE;
				END_IF
			END_IF

			(* close off fbCloseAllPorts *)
			fbCloseAllPorts(bExecute := FALSE);
		END_IF


	(* complete *)
	E_TCPIP_DONE:

		(* update outputs *)
		bBusy := FALSE;
		bDone := TRUE;

		eState := E_TCPIP_IDLE;


